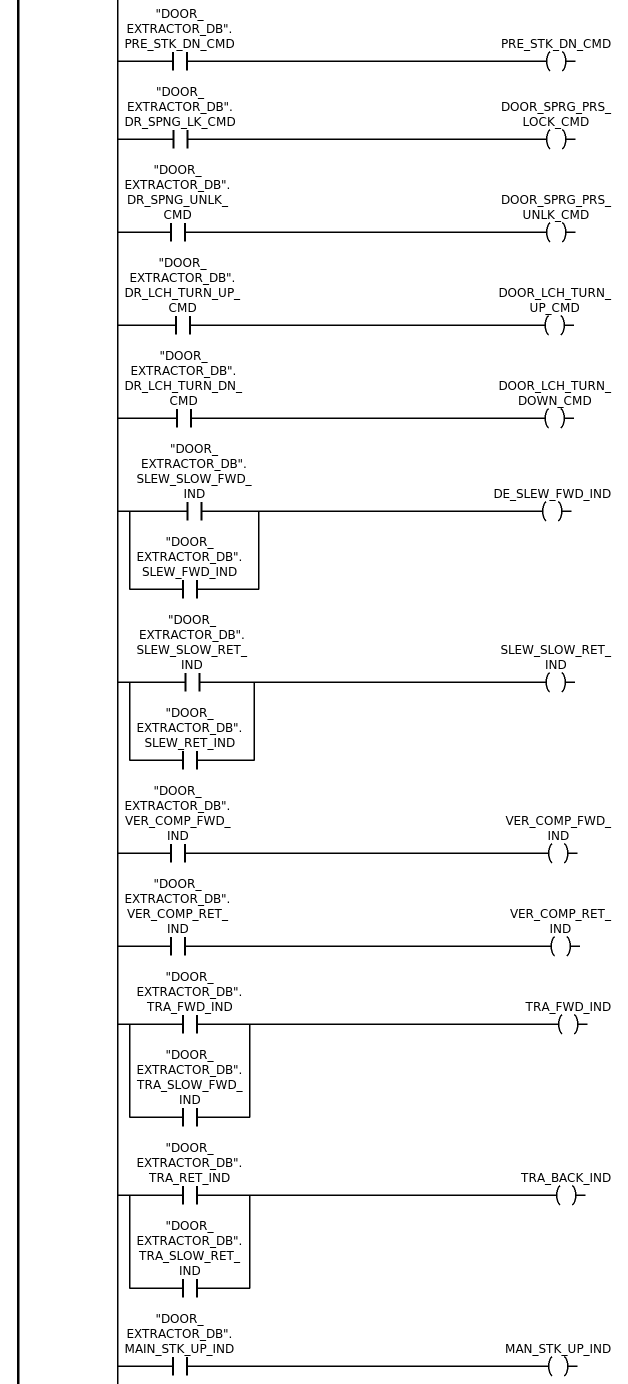
[picture p48: OUTPUT_MAPPING networks 12-12]
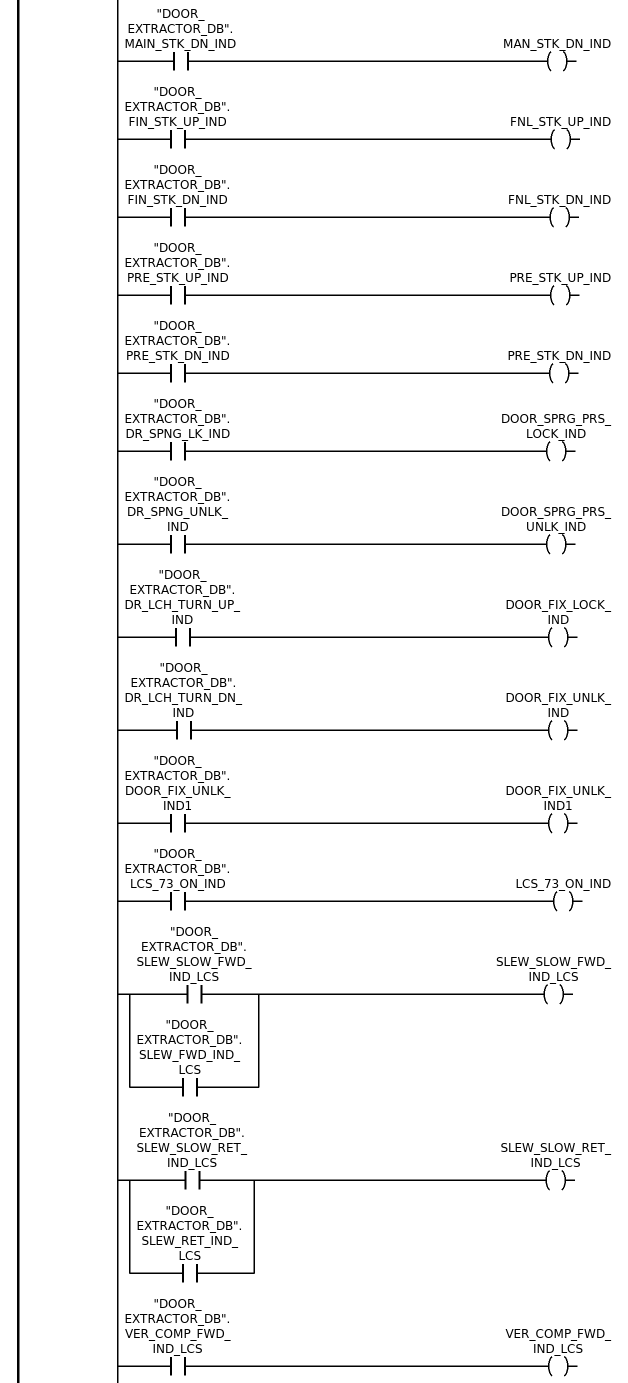
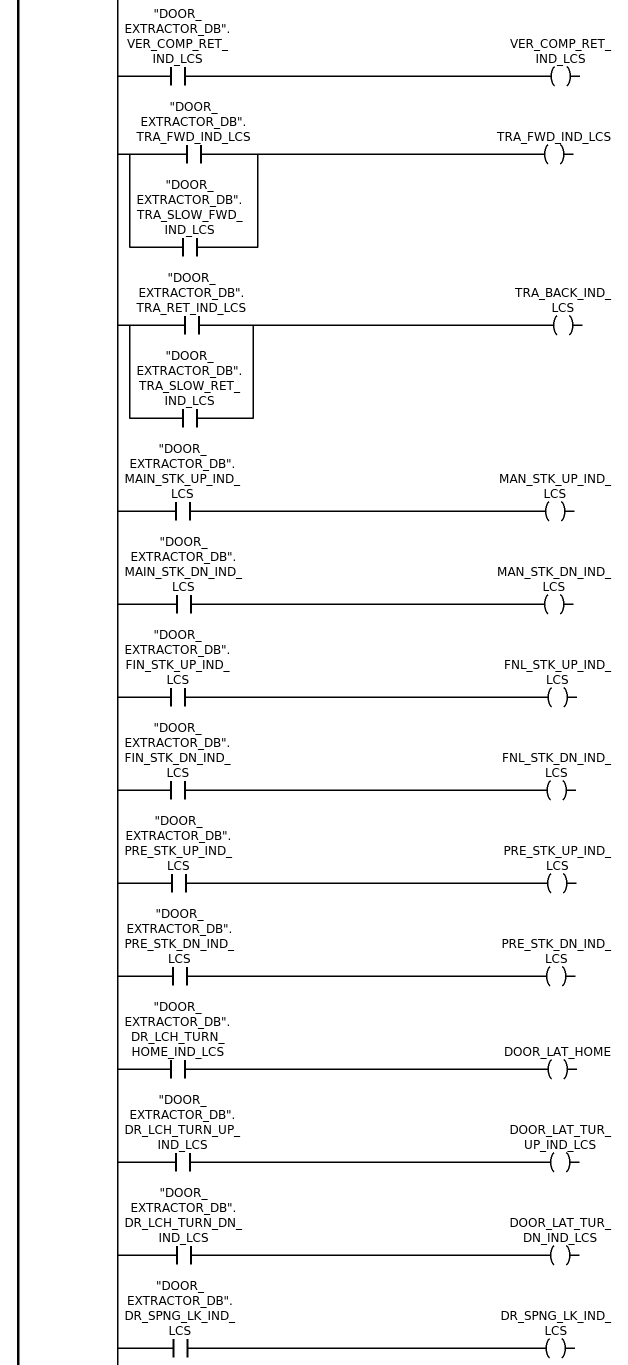
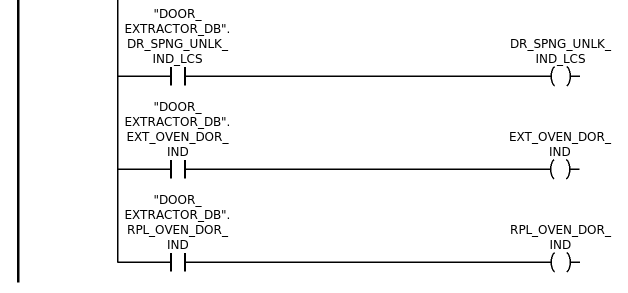
NETWORK
TITLE =
      A     "ALWAYS_ON";
      =     L 0.0;
      A     L 0.0;
      A     "DOOR_EXTRACTOR_DB".SLEW_NOR_FWD_COMMAND;
      =     "SLEW_NOR_FWD_COMMAND";
      A     L 0.0;
      A     "DOOR_EXTRACTOR_DB".SLEW_NOR_RET_COMMAND;
      =     "SLEW_NOR_RET_COMMAND";
      A     L 0.0;
      A     "DOOR_EXTRACTOR_DB".VER_COMP_FWD_CMD;
      =     "VER_COMP_FWD_CMD";
      A     L 0.0;
      A     "DOOR_EXTRACTOR_DB".VER_COMP_RET_CMD;
      =     "VER_COMP_RET_CMD";
      A     L 0.0;
      A     "DOOR_EXTRACTOR_DB".VER_COMP_RELIVE_CMD;
      =     "VER_COMP_RELIVE_CMD";
      A     L 0.0;
      A     "DOOR_EXTRACTOR_DB".TRA_SLOW_FWD_CMD;
      =     "TRA_SLOW_FWD_CMD";
      A     L 0.0;
      A     "DOOR_EXTRACTOR_DB".TRA_SLOW_RET_CMD;
      =     "TRA_SLOW_RET_CMD";
      A     L 0.0;
      A     "DOOR_EXTRACTOR_DB".TRA_NOR_FWD_CMD;
      =     "TRA_NORM_FWD_CMD";
      A     L 0.0;
      A     "DOOR_EXTRACTOR_DB".TRA_NOR_RET_CMD;
      =     "TRA_NORM_RET_CMD";
      A     L 0.0;
      A     "DOOR_EXTRACTOR_DB".TRA_RELIVE_CMD;
      =     "DE_TRA_RELIVE_CMD";
      A     L 0.0;
      A(;
      O     "DOOR_EXTRACTOR_DB".MAIN_STK_UP_CMD;
      O     "DOOR_EXTRACTOR_DB".FIN_STK_UP_CMD;
      );
      =     "MAN_FNL_STK_UP_CMD";
      A     L 0.0;
      A(;
      O     "DOOR_EXTRACTOR_DB".MAIN_STK_DN_CMD;
      O     "DOOR_EXTRACTOR_DB".FIN_STK_DN_CMD;
      );
      =     "MAN_FNL_STK_DN_CMD";
      A     L 0.0;
      A     "DOOR_EXTRACTOR_DB".PRE_STK_UP_CMD;
      =     "PRE_STK_UP_CMD";
      A     L 0.0;
      A     "DOOR_EXTRACTOR_DB".PRE_STK_DN_CMD;
      =     "PRE_STK_DN_CMD";
      A     L 0.0;
      A     "DOOR_EXTRACTOR_DB".DR_SPNG_LK_CMD;
      =     "DOOR_SPRG_PRS_LOCK_CMD";
      A     L 0.0;
      A     "DOOR_EXTRACTOR_DB".DR_SPNG_UNLK_CMD;
      =     "DOOR_SPRG_PRS_UNLK_CMD";
      A     L 0.0;
      A     "DOOR_EXTRACTOR_DB".DR_LCH_TURN_UP_CMD;
      =     "DOOR_LCH_TURN_UP_CMD";
      A     L 0.0;
      A     "DOOR_EXTRACTOR_DB".DR_LCH_TURN_DN_CMD;
      =     "DOOR_LCH_TURN_DOWN_CMD";
      A     L 0.0;
      A(;
      O     "DOOR_EXTRACTOR_DB".SLEW_SLOW_FWD_IND;
      O     "DOOR_EXTRACTOR_DB".SLEW_FWD_IND;
      );
      =     "DE_SLEW_FWD_IND";
      A     L 0.0;
      A(;
      O     "DOOR_EXTRACTOR_DB".SLEW_SLOW_RET_IND;
      O     "DOOR_EXTRACTOR_DB".SLEW_RET_IND;
      );
      =     "SLEW_SLOW_RET_IND";
      A     L 0.0;
      A     "DOOR_EXTRACTOR_DB".VER_COMP_FWD_IND;
      =     "VER_COMP_FWD_IND";
      A     L 0.0;
      A     "DOOR_EXTRACTOR_DB".VER_COMP_RET_IND;
      =     "VER_COMP_RET_IND";
      A     L 0.0;
      A(;
      O     "DOOR_EXTRACTOR_DB".TRA_FWD_IND;
      O     "DOOR_EXTRACTOR_DB".TRA_SLOW_FWD_IND;
      );
      =     "TRA_FWD_IND";
      A     L 0.0;
      A(;
      O     "DOOR_EXTRACTOR_DB".TRA_RET_IND;
      O     "DOOR_EXTRACTOR_DB".TRA_SLOW_RET_IND;
      );
      =     "TRA_BACK_IND";
      A     L 0.0;
      A     "DOOR_EXTRACTOR_DB".MAIN_STK_UP_IND;
      =     "MAN_STK_UP_IND";
      A     L 0.0;
      A     "DOOR_EXTRACTOR_DB".MAIN_STK_DN_IND;
      =     "MAN_STK_DN_IND";
      A     L 0.0;
      A     "DOOR_EXTRACTOR_DB".FIN_STK_UP_IND;
      =     "FNL_STK_UP_IND";
      A     L 0.0;
      A     "DOOR_EXTRACTOR_DB".FIN_STK_DN_IND;
      =     "FNL_STK_DN_IND";
      A     L 0.0;
      A     "DOOR_EXTRACTOR_DB".PRE_STK_UP_IND;
      =     "PRE_STK_UP_IND";
      A     L 0.0;
      A     "DOOR_EXTRACTOR_DB".PRE_STK_DN_IND;
      =     "PRE_STK_DN_IND";
      A     L 0.0;
      A     "DOOR_EXTRACTOR_DB".DR_SPNG_LK_IND;
      =     "DOOR_SPRG_PRS_LOCK_IND";
      A     L 0.0;
      A     "DOOR_EXTRACTOR_DB".DR_SPNG_UNLK_IND;
      =     "DOOR_SPRG_PRS_UNLK_IND";
      A     L 0.0;
      A     "DOOR_EXTRACTOR_DB".DR_LCH_TURN_UP_IND;
      =     "DOOR_FIX_LOCK_IND";
      A     L 0.0;
      A     "DOOR_EXTRACTOR_DB".DR_LCH_TURN_DN_IND;
      =     "DOOR_FIX_UNLK_IND";
      A     L 0.0;
      A     "DOOR_EXTRACTOR_DB".DOOR_FIX_UNLK_IND1;
      =     "DOOR_FIX_UNLK_IND1";
      A     L 0.0;
      A     "DOOR_EXTRACTOR_DB".LCS_73_ON_IND;
      =     "LCS_73_ON_IND";
      A     L 0.0;
      A(;
      O     "DOOR_EXTRACTOR_DB".SLEW_SLOW_FWD_IND_LCS;
      O     "DOOR_EXTRACTOR_DB".SLEW_FWD_IND_LCS;
      );
      =     "SLEW_SLOW_FWD_IND_LCS";
      A     L 0.0;
      A(;
      O     "DOOR_EXTRACTOR_DB".SLEW_SLOW_RET_IND_LCS;
      O     "DOOR_EXTRACTOR_DB".SLEW_RET_IND_LCS;
      );
      =     "SLEW_SLOW_RET_IND_LCS";
      A     L 0.0;
      A     "DOOR_EXTRACTOR_DB".VER_COMP_FWD_IND_LCS;
      =     "VER_COMP_FWD_IND_LCS";
      A     L 0.0;
      A     "DOOR_EXTRACTOR_DB".VER_COMP_RET_IND_LCS;
      =     "VER_COMP_RET_IND_LCS";
      A     L 0.0;
      A(;
      O     "DOOR_EXTRACTOR_DB".TRA_FWD_IND_LCS;
      O     "DOOR_EXTRACTOR_DB".TRA_SLOW_FWD_IND_LCS;
      );
      =     "TRA_FWD_IND_LCS";
      A     L 0.0;
      A(;
      O     "DOOR_EXTRACTOR_DB".TRA_RET_IND_LCS;
      O     "DOOR_EXTRACTOR_DB".TRA_SLOW_RET_IND_LCS;
      );
      =     "TRA_BACK_IND_LCS";
      A     L 0.0;
      A     "DOOR_EXTRACTOR_DB".MAIN_STK_UP_IND_LCS;
      =     "MAN_STK_UP_IND_LCS";
      A     L 0.0;
      A     "DOOR_EXTRACTOR_DB".MAIN_STK_DN_IND_LCS;
      =     "MAN_STK_DN_IND_LCS";
      A     L 0.0;
      A     "DOOR_EXTRACTOR_DB".FIN_STK_UP_IND_LCS;
      =     "FNL_STK_UP_IND_LCS";
      A     L 0.0;
      A     "DOOR_EXTRACTOR_DB".FIN_STK_DN_IND_LCS;
      =     "FNL_STK_DN_IND_LCS";
      A     L 0.0;
      A     "DOOR_EXTRACTOR_DB".PRE_STK_UP_IND_LCS;
      =     "PRE_STK_UP_IND_LCS";
      A     L 0.0;
      A     "DOOR_EXTRACTOR_DB".PRE_STK_DN_IND_LCS;
      =     "PRE_STK_DN_IND_LCS";
      A     L 0.0;
      A     "DOOR_EXTRACTOR_DB".DR_LCH_TURN_HOME_IND_LCS;
      =     "DOOR_LAT_HOME";
      A     L 0.0;
      A     "DOOR_EXTRACTOR_DB".DR_LCH_TURN_UP_IND_LCS;
      =     "DOOR_LAT_TUR_UP_IND_LCS";
      A     L 0.0;
      A     "DOOR_EXTRACTOR_DB".DR_LCH_TURN_DN_IND_LCS;
      =     "DOOR_LAT_TUR_DN_IND_LCS";
      A     L 0.0;
      A     "DOOR_EXTRACTOR_DB".DR_SPNG_LK_IND_LCS;
      =     "DR_SPNG_LK_IND_LCS";
      A     L 0.0;
      A     "DOOR_EXTRACTOR_DB".DR_SPNG_UNLK_IND_LCS;
      =     "DR_SPNG_UNLK_IND_LCS";
      A     L 0.0;
      A     "DOOR_EXTRACTOR_DB".EXT_OVEN_DOR_IND;
      =     "EXT_OVEN_DOR_IND";
      A     L 0.0;
      A     "DOOR_EXTRACTOR_DB".RPL_OVEN_DOR_IND;
      =     "RPL_OVEN_DOR_IND";
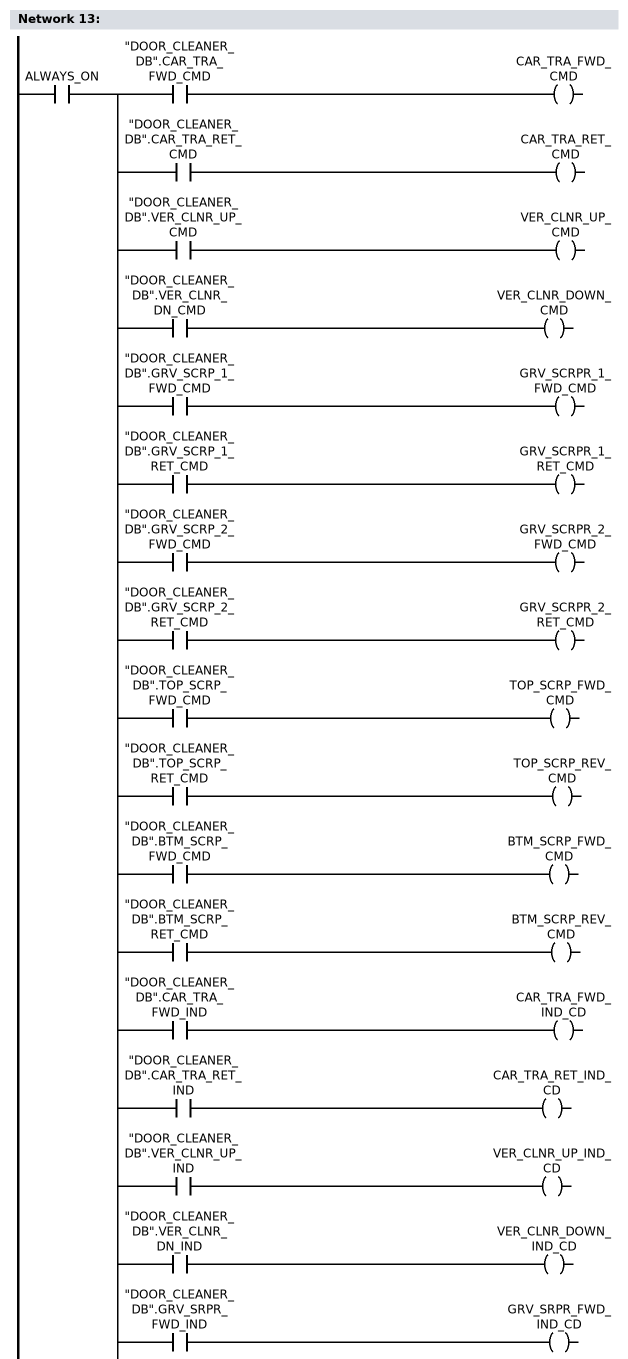
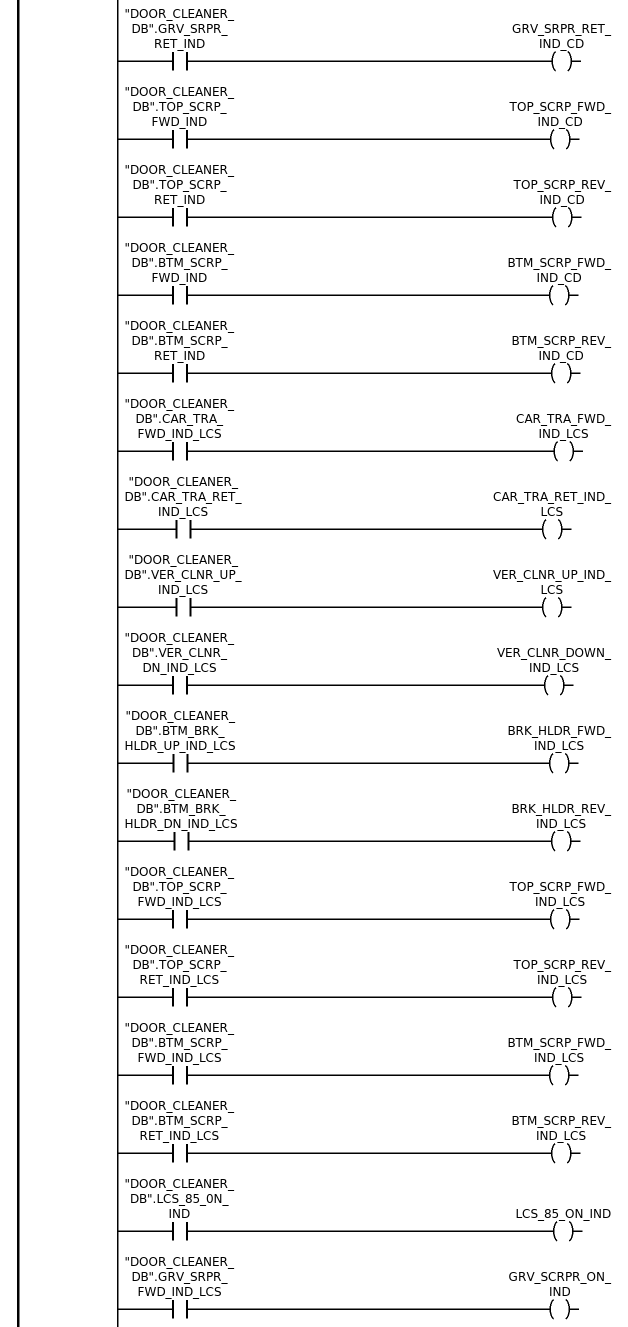
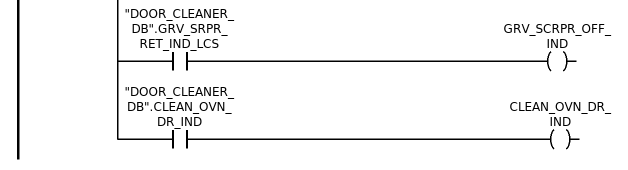
NETWORK
TITLE =
      A     "ALWAYS_ON";
      =     L 0.0;
      A     L 0.0;
      A     "DOOR_CLEANER_DB".CAR_TRA_FWD_CMD;
      =     "CAR_TRA_FWD_CMD";
      A     L 0.0;
      A     "DOOR_CLEANER_DB".CAR_TRA_RET_CMD;
      =     "CAR_TRA_RET_CMD";
      A     L 0.0;
      A     "DOOR_CLEANER_DB".VER_CLNR_UP_CMD;
      =     "VER_CLNR_UP_CMD";
      A     L 0.0;
      A     "DOOR_CLEANER_DB".VER_CLNR_DN_CMD;
      =     "VER_CLNR_DOWN_CMD";
      A     L 0.0;
      A     "DOOR_CLEANER_DB".GRV_SCRP_1_FWD_CMD;
      =     "GRV_SCRPR_1_FWD_CMD";
      A     L 0.0;
      A     "DOOR_CLEANER_DB".GRV_SCRP_1_RET_CMD;
      =     "GRV_SCRPR_1_RET_CMD";
      A     L 0.0;
      A     "DOOR_CLEANER_DB".GRV_SCRP_2_FWD_CMD;
      =     "GRV_SCRPR_2_FWD_CMD";
      A     L 0.0;
      A     "DOOR_CLEANER_DB".GRV_SCRP_2_RET_CMD;
      =     "GRV_SCRPR_2_RET_CMD";
      A     L 0.0;
      A     "DOOR_CLEANER_DB".TOP_SCRP_FWD_CMD;
      =     "TOP_SCRP_FWD_CMD";
      A     L 0.0;
      A     "DOOR_CLEANER_DB".TOP_SCRP_RET_CMD;
      =     "TOP_SCRP_REV_CMD";
      A     L 0.0;
      A     "DOOR_CLEANER_DB".BTM_SCRP_FWD_CMD;
      =     "BTM_SCRP_FWD_CMD";
      A     L 0.0;
      A     "DOOR_CLEANER_DB".BTM_SCRP_RET_CMD;
      =     "BTM_SCRP_REV_CMD";
      A     L 0.0;
      A     "DOOR_CLEANER_DB".CAR_TRA_FWD_IND;
      =     "CAR_TRA_FWD_IND_CD";
      A     L 0.0;
      A     "DOOR_CLEANER_DB".CAR_TRA_RET_IND;
      =     "CAR_TRA_RET_IND_CD";
      A     L 0.0;
      A     "DOOR_CLEANER_DB".VER_CLNR_UP_IND;
      =     "VER_CLNR_UP_IND_CD";
      A     L 0.0;
      A     "DOOR_CLEANER_DB".VER_CLNR_DN_IND;
      =     "VER_CLNR_DOWN_IND_CD";
      A     L 0.0;
      A     "DOOR_CLEANER_DB".GRV_SRPR_FWD_IND;
      =     "GRV_SRPR_FWD_IND_CD";
      A     L 0.0;
      A     "DOOR_CLEANER_DB".GRV_SRPR_RET_IND;
      =     "GRV_SRPR_RET_IND_CD";
      A     L 0.0;
      A     "DOOR_CLEANER_DB".TOP_SCRP_FWD_IND;
      =     "TOP_SCRP_FWD_IND_CD";
      A     L 0.0;
      A     "DOOR_CLEANER_DB".TOP_SCRP_RET_IND;
      =     "TOP_SCRP_REV_IND_CD";
      A     L 0.0;
      A     "DOOR_CLEANER_DB".BTM_SCRP_FWD_IND;
      =     "BTM_SCRP_FWD_IND_CD";
      A     L 0.0;
      A     "DOOR_CLEANER_DB".BTM_SCRP_RET_IND;
      =     "BTM_SCRP_REV_IND_CD";
      A     L 0.0;
      A     "DOOR_CLEANER_DB".CAR_TRA_FWD_IND_LCS;
      =     "CAR_TRA_FWD_IND_LCS";
      A     L 0.0;
      A     "DOOR_CLEANER_DB".CAR_TRA_RET_IND_LCS;
      =     "CAR_TRA_RET_IND_LCS";
      A     L 0.0;
      A     "DOOR_CLEANER_DB".VER_CLNR_UP_IND_LCS;
      =     "VER_CLNR_UP_IND_LCS";
      A     L 0.0;
      A     "DOOR_CLEANER_DB".VER_CLNR_DN_IND_LCS;
      =     "VER_CLNR_DOWN_IND_LCS";
      A     L 0.0;
      A     "DOOR_CLEANER_DB".BTM_BRK_HLDR_UP_IND_LCS;
      =     "BRK_HLDR_FWD_IND_LCS";
      A     L 0.0;
      A     "DOOR_CLEANER_DB".BTM_BRK_HLDR_DN_IND_LCS;
      =     "BRK_HLDR_REV_IND_LCS";
      A     L 0.0;
      A     "DOOR_CLEANER_DB".TOP_SCRP_FWD_IND_LCS;
      =     "TOP_SCRP_FWD_IND_LCS";
      A     L 0.0;
      A     "DOOR_CLEANER_DB".TOP_SCRP_RET_IND_LCS;
      =     "TOP_SCRP_REV_IND_LCS";
      A     L 0.0;
      A     "DOOR_CLEANER_DB".BTM_SCRP_FWD_IND_LCS;
      =     "BTM_SCRP_FWD_IND_LCS";
      A     L 0.0;
      A     "DOOR_CLEANER_DB".BTM_SCRP_RET_IND_LCS;
      =     "BTM_SCRP_REV_IND_LCS";
      A     L 0.0;
      A     "DOOR_CLEANER_DB".LCS_85_0N_IND;
      =     "LCS_85_ON_IND";
      A     L 0.0;
      A     "DOOR_CLEANER_DB".GRV_SRPR_FWD_IND_LCS;
      =     "GRV_SCRPR_ON_IND";
      A     L 0.0;
      A     "DOOR_CLEANER_DB".GRV_SRPR_RET_IND_LCS;
      =     "GRV_SCRPR_OFF_IND";
      A     L 0.0;
      A     "DOOR_CLEANER_DB".CLEAN_OVN_DR_IND;
      =     "CLEAN_OVN_DR_IND";
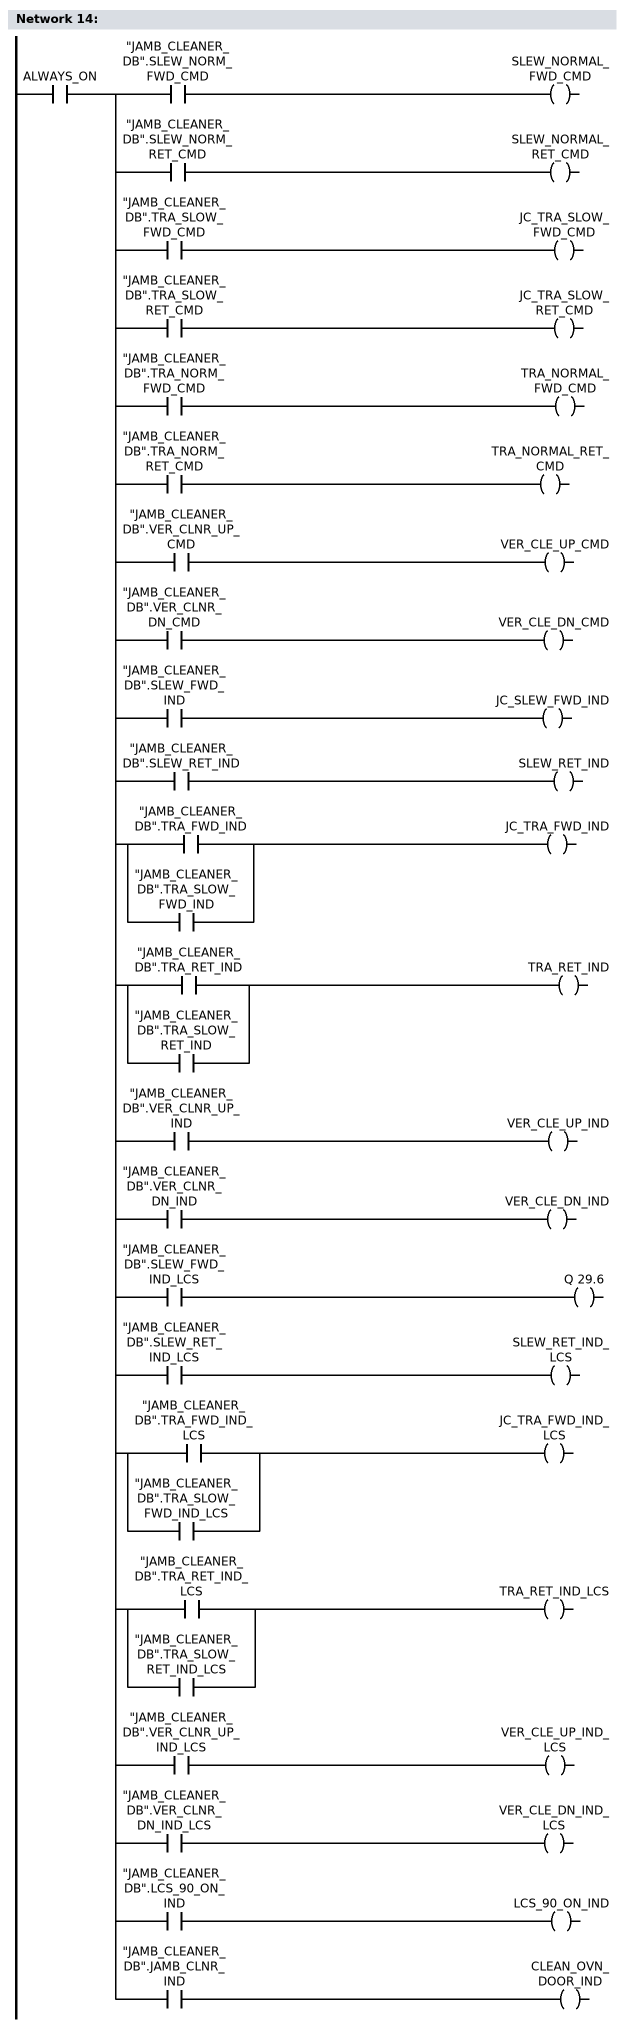
NETWORK
TITLE =
      A     "ALWAYS_ON";
      =     L 0.0;
      A     L 0.0;
      A     "JAMB_CLEANER_DB".SLEW_NORM_FWD_CMD;
      =     "SLEW_NORMAL_FWD_CMD";
      A     L 0.0;
      A     "JAMB_CLEANER_DB".SLEW_NORM_RET_CMD;
      =     "SLEW_NORMAL_RET_CMD";
      A     L 0.0;
      A     "JAMB_CLEANER_DB".TRA_SLOW_FWD_CMD;
      =     "JC_TRA_SLOW_FWD_CMD";
      A     L 0.0;
      A     "JAMB_CLEANER_DB".TRA_SLOW_RET_CMD;
      =     "JC_TRA_SLOW_RET_CMD";
      A     L 0.0;
      A     "JAMB_CLEANER_DB".TRA_NORM_FWD_CMD;
      =     "TRA_NORMAL_FWD_CMD";
      A     L 0.0;
      A     "JAMB_CLEANER_DB".TRA_NORM_RET_CMD;
      =     "TRA_NORMAL_RET_CMD";
      A     L 0.0;
      A     "JAMB_CLEANER_DB".VER_CLNR_UP_CMD;
      =     "VER_CLE_UP_CMD";
      A     L 0.0;
      A     "JAMB_CLEANER_DB".VER_CLNR_DN_CMD;
      =     "VER_CLE_DN_CMD";
      A     L 0.0;
      A     "JAMB_CLEANER_DB".SLEW_FWD_IND;
      =     "JC_SLEW_FWD_IND";
      A     L 0.0;
      A     "JAMB_CLEANER_DB".SLEW_RET_IND;
      =     "SLEW_RET_IND";
      A     L 0.0;
      A(;
      O     "JAMB_CLEANER_DB".TRA_FWD_IND;
      O     "JAMB_CLEANER_DB".TRA_SLOW_FWD_IND;
      );
      =     "JC_TRA_FWD_IND";
      A     L 0.0;
      A(;
      O     "JAMB_CLEANER_DB".TRA_RET_IND;
      O     "JAMB_CLEANER_DB".TRA_SLOW_RET_IND;
      );
      =     "TRA_RET_IND";
      A     L 0.0;
      A     "JAMB_CLEANER_DB".VER_CLNR_UP_IND;
      =     "VER_CLE_UP_IND";
      A     L 0.0;
      A     "JAMB_CLEANER_DB".VER_CLNR_DN_IND;
      =     "VER_CLE_DN_IND";
      A     L 0.0;
      A     "JAMB_CLEANER_DB".SLEW_FWD_IND_LCS;
      =     Q 29.6;
      A     L 0.0;
      A     "JAMB_CLEANER_DB".SLEW_RET_IND_LCS;
      =     "SLEW_RET_IND_LCS";
      A     L 0.0;
      A(;
      O     "JAMB_CLEANER_DB".TRA_FWD_IND_LCS;
      O     "JAMB_CLEANER_DB".TRA_SLOW_FWD_IND_LCS;
      );
      =     "JC_TRA_FWD_IND_LCS";
      A     L 0.0;
      A(;
      O     "JAMB_CLEANER_DB".TRA_RET_IND_LCS;
      O     "JAMB_CLEANER_DB".TRA_SLOW_RET_IND_LCS;
      );
      =     "TRA_RET_IND_LCS";
      A     L 0.0;
      A     "JAMB_CLEANER_DB".VER_CLNR_UP_IND_LCS;
      =     "VER_CLE_UP_IND_LCS";
      A     L 0.0;
      A     "JAMB_CLEANER_DB".VER_CLNR_DN_IND_LCS;
      =     "VER_CLE_DN_IND_LCS";
      A     L 0.0;
      A     "JAMB_CLEANER_DB".LCS_90_ON_IND;
      =     "LCS_90_ON_IND";
      A     L 0.0;
      A     "JAMB_CLEANER_DB".JAMB_CLNR_IND;
      =     "CLEAN_OVN_DOOR_IND";
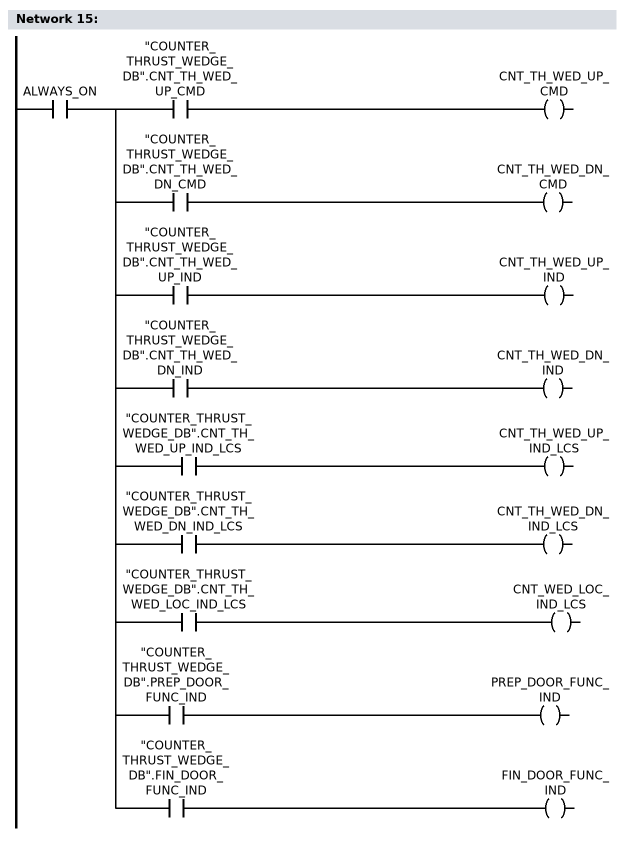
NETWORK
TITLE =
      A     "ALWAYS_ON";
      =     L 0.0;
      A     L 0.0;
      A     "COUNTER_THRUST_WEDGE_DB".CNT_TH_WED_UP_CMD;
      =     "CNT_TH_WED_UP_CMD";
      A     L 0.0;
      A     "COUNTER_THRUST_WEDGE_DB".CNT_TH_WED_DN_CMD;
      =     "CNT_TH_WED_DN_CMD";
      A     L 0.0;
      A     "COUNTER_THRUST_WEDGE_DB".CNT_TH_WED_UP_IND;
      =     "CNT_TH_WED_UP_IND";
      A     L 0.0;
      A     "COUNTER_THRUST_WEDGE_DB".CNT_TH_WED_DN_IND;
      =     "CNT_TH_WED_DN_IND";
      A     L 0.0;
      A     "COUNTER_THRUST_WEDGE_DB".CNT_TH_WED_UP_IND_LCS;
      =     "CNT_TH_WED_UP_IND_LCS";
      A     L 0.0;
      A     "COUNTER_THRUST_WEDGE_DB".CNT_TH_WED_DN_IND_LCS;
      =     "CNT_TH_WED_DN_IND_LCS";
      A     L 0.0;
      A     "COUNTER_THRUST_WEDGE_DB".CNT_TH_WED_LOC_IND_LCS;
      =     "CNT_WED_LOC_IND_LCS";
      A     L 0.0;
      A     "COUNTER_THRUST_WEDGE_DB".PREP_DOOR_FUNC_IND;
      =     "PREP_DOOR_FUNC_IND";
      A     L 0.0;
      A     "COUNTER_THRUST_WEDGE_DB".FIN_DOOR_FUNC_IND;
      =     "FIN_DOOR_FUNC_IND";
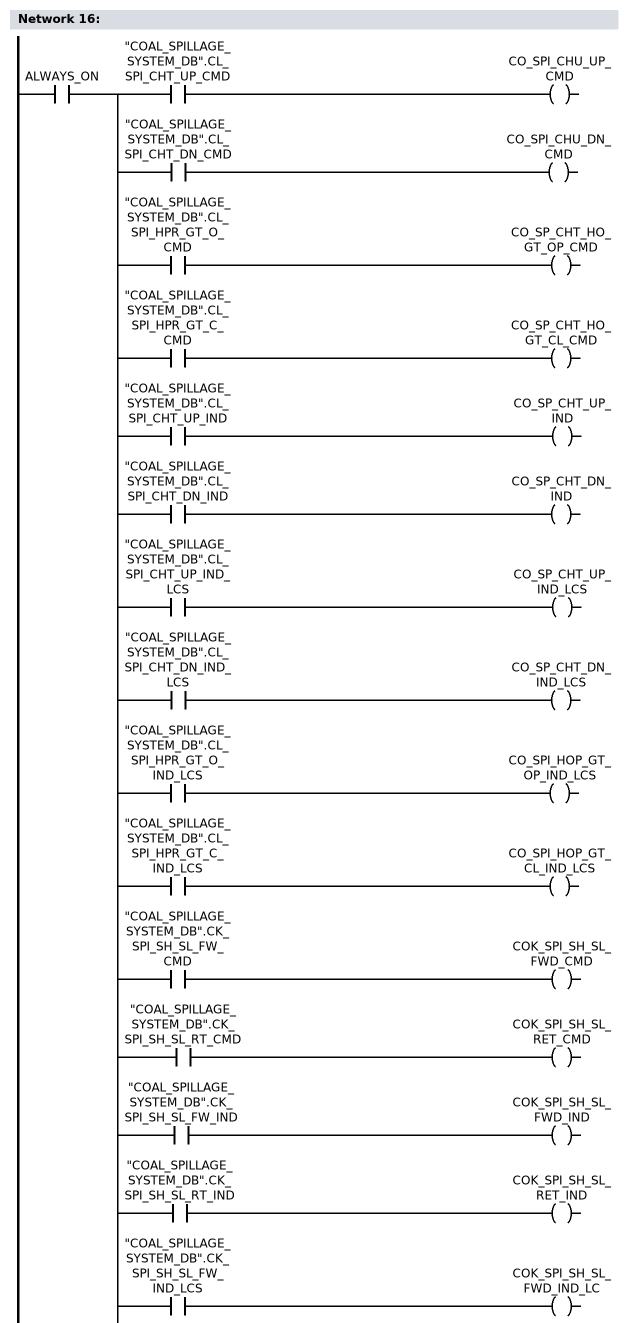
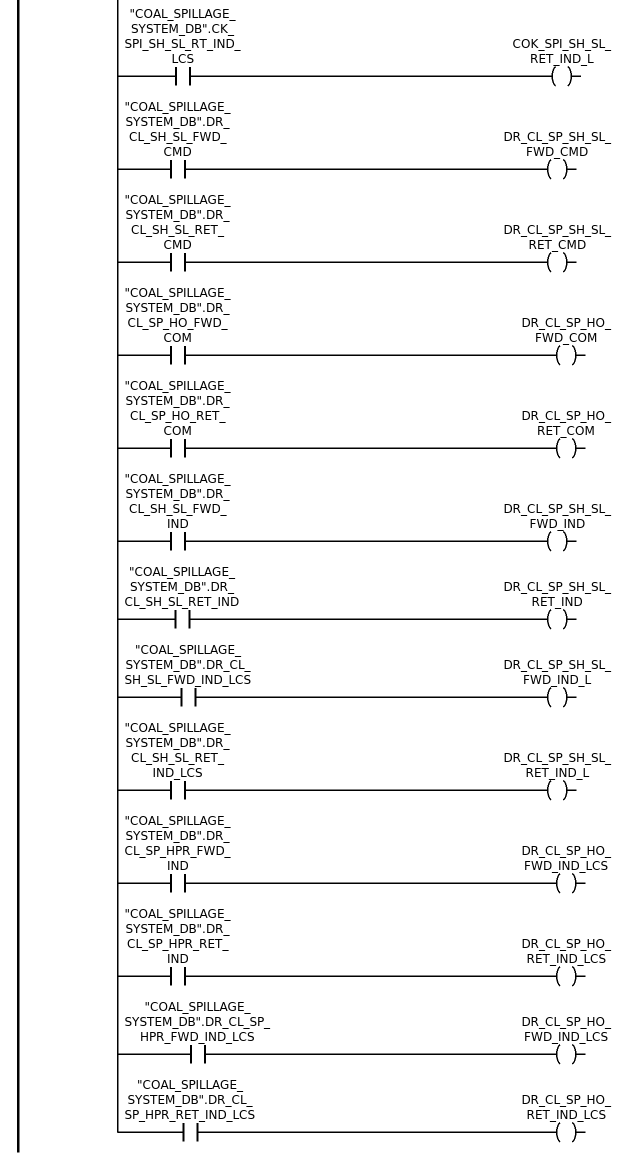
NETWORK
TITLE =
      A     "ALWAYS_ON";
      =     L 0.0;
      A     L 0.0;
      A     "COAL_SPILLAGE_SYSTEM_DB".CL_SPI_CHT_UP_CMD;
      =     "CO_SPI_CHU_UP_CMD";
      A     L 0.0;
      A     "COAL_SPILLAGE_SYSTEM_DB".CL_SPI_CHT_DN_CMD;
      =     "CO_SPI_CHU_DN_CMD";
      A     L 0.0;
      A     "COAL_SPILLAGE_SYSTEM_DB".CL_SPI_HPR_GT_O_CMD;
      =     "CO_SP_CHT_HO_GT_OP_CMD";
      A     L 0.0;
      A     "COAL_SPILLAGE_SYSTEM_DB".CL_SPI_HPR_GT_C_CMD;
      =     "CO_SP_CHT_HO_GT_CL_CMD";
      A     L 0.0;
      A     "COAL_SPILLAGE_SYSTEM_DB".CL_SPI_CHT_UP_IND;
      =     "CO_SP_CHT_UP_IND";
      A     L 0.0;
      A     "COAL_SPILLAGE_SYSTEM_DB".CL_SPI_CHT_DN_IND;
      =     "CO_SP_CHT_DN_IND";
      A     L 0.0;
      A     "COAL_SPILLAGE_SYSTEM_DB".CL_SPI_CHT_UP_IND_LCS;
      =     "CO_SP_CHT_UP_IND_LCS";
      A     L 0.0;
      A     "COAL_SPILLAGE_SYSTEM_DB".CL_SPI_CHT_DN_IND_LCS;
      =     "CO_SP_CHT_DN_IND_LCS";
      A     L 0.0;
      A     "COAL_SPILLAGE_SYSTEM_DB".CL_SPI_HPR_GT_O_IND_LCS;
      =     "CO_SPI_HOP_GT_OP_IND_LCS";
      A     L 0.0;
      A     "COAL_SPILLAGE_SYSTEM_DB".CL_SPI_HPR_GT_C_IND_LCS;
      =     "CO_SPI_HOP_GT_CL_IND_LCS";
      A     L 0.0;
      A     "COAL_SPILLAGE_SYSTEM_DB".CK_SPI_SH_SL_FW_CMD;
      =     "COK_SPI_SH_SL_FWD_CMD";
      A     L 0.0;
      A     "COAL_SPILLAGE_SYSTEM_DB".CK_SPI_SH_SL_RT_CMD;
      =     "COK_SPI_SH_SL_RET_CMD";
      A     L 0.0;
      A     "COAL_SPILLAGE_SYSTEM_DB".CK_SPI_SH_SL_FW_IND;
      =     "COK_SPI_SH_SL_FWD_IND";
      A     L 0.0;
      A     "COAL_SPILLAGE_SYSTEM_DB".CK_SPI_SH_SL_RT_IND;
      =     "COK_SPI_SH_SL_RET_IND";
      A     L 0.0;
      A     "COAL_SPILLAGE_SYSTEM_DB".CK_SPI_SH_SL_FW_IND_LCS;
      =     "COK_SPI_SH_SL_FWD_IND_LC";
      A     L 0.0;
      A     "COAL_SPILLAGE_SYSTEM_DB".CK_SPI_SH_SL_RT_IND_LCS;
      =     "COK_SPI_SH_SL_RET_IND_L";
      A     L 0.0;
      A     "COAL_SPILLAGE_SYSTEM_DB".DR_CL_SH_SL_FWD_CMD;
      =     "DR_CL_SP_SH_SL_FWD_CMD";
      A     L 0.0;
      A     "COAL_SPILLAGE_SYSTEM_DB".DR_CL_SH_SL_RET_CMD;
      =     "DR_CL_SP_SH_SL_RET_CMD";
      A     L 0.0;
      A     "COAL_SPILLAGE_SYSTEM_DB".DR_CL_SP_HO_FWD_COM;
      =     "DR_CL_SP_HO_FWD_COM";
      A     L 0.0;
      A     "COAL_SPILLAGE_SYSTEM_DB".DR_CL_SP_HO_RET_COM;
      =     "DR_CL_SP_HO_RET_COM";
      A     L 0.0;
      A     "COAL_SPILLAGE_SYSTEM_DB".DR_CL_SH_SL_FWD_IND;
      =     "DR_CL_SP_SH_SL_FWD_IND";
      A     L 0.0;
      A     "COAL_SPILLAGE_SYSTEM_DB".DR_CL_SH_SL_RET_IND;
      =     "DR_CL_SP_SH_SL_RET_IND";
      A     L 0.0;
      A     "COAL_SPILLAGE_SYSTEM_DB".DR_CL_SH_SL_FWD_IND_LCS;
      =     "DR_CL_SP_SH_SL_FWD_IND_L";
      A     L 0.0;
      A     "COAL_SPILLAGE_SYSTEM_DB".DR_CL_SH_SL_RET_IND_LCS;
      =     "DR_CL_SP_SH_SL_RET_IND_L";
      A     L 0.0;
      A     "COAL_SPILLAGE_SYSTEM_DB".DR_CL_SP_HPR_FWD_IND;
      =     "DR_CL_SP_HO_FWD_IND_LCS";
      A     L 0.0;
      A     "COAL_SPILLAGE_SYSTEM_DB".DR_CL_SP_HPR_RET_IND;
      =     "DR_CL_SP_HO_RET_IND_LCS";
      A     L 0.0;
      A     "COAL_SPILLAGE_SYSTEM_DB".DR_CL_SP_HPR_FWD_IND_LCS;
      =     "DR_CL_SP_HO_FWD_IND_LCS";
      A     L 0.0;
      A     "COAL_SPILLAGE_SYSTEM_DB".DR_CL_SP_HPR_RET_IND_LCS;
      =     "DR_CL_SP_HO_RET_IND_LCS";
END_FUNCTION

FUNCTION "MAIN_POWER" : VOID	// FC 3
AUTHOR : Kamillas
VERSION : 0.1
BEGIN
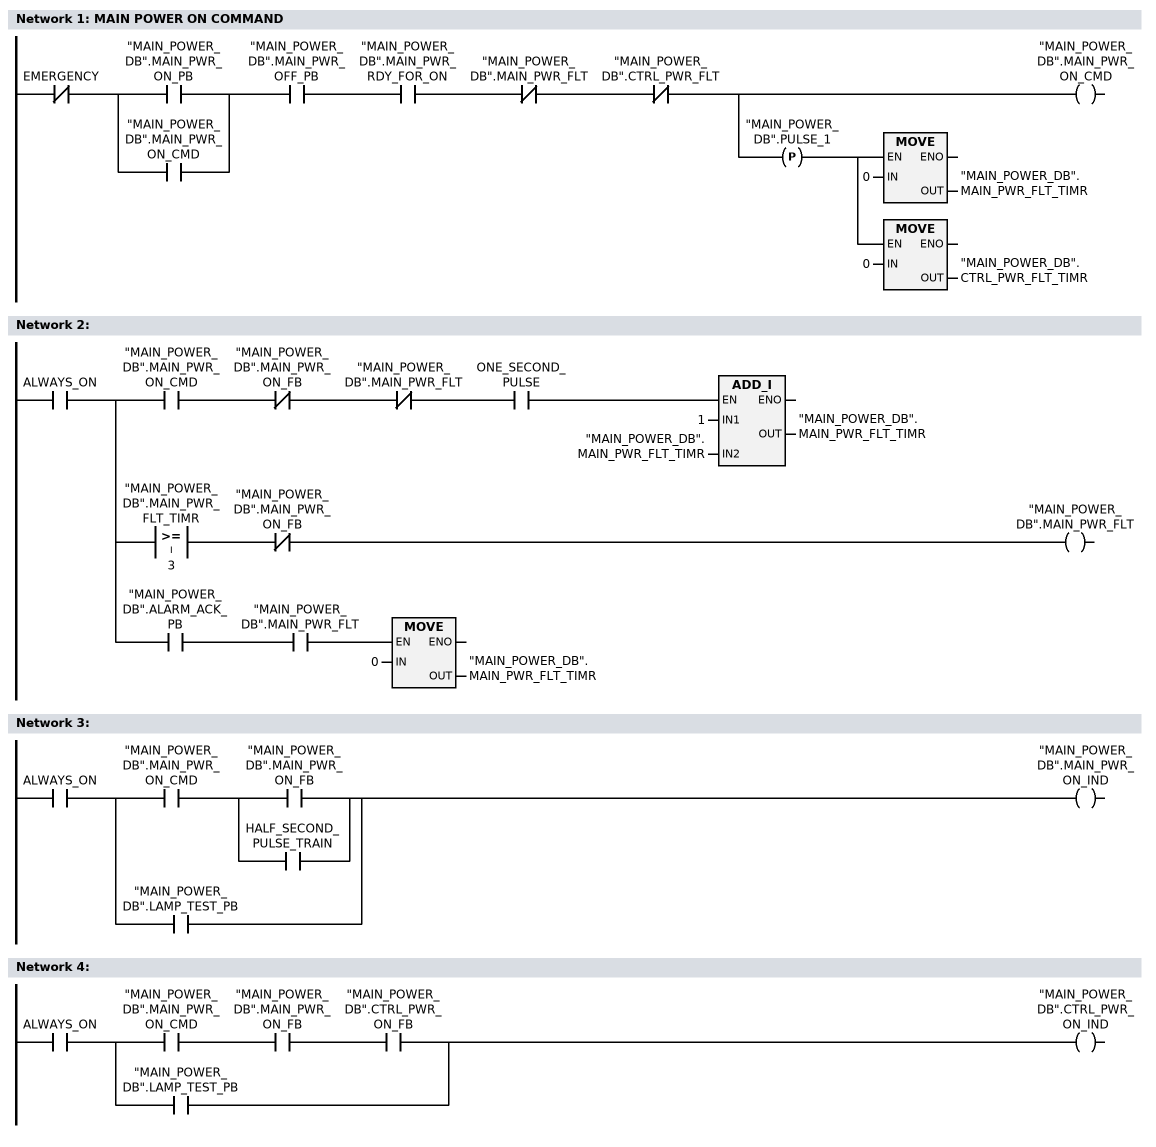
NETWORK
TITLE = MAIN POWER ON COMMAND
      AN    "EMERGENCY";
      A(;
      O     "MAIN_POWER_DB".MAIN_PWR_ON_PB;
      O     "MAIN_POWER_DB".MAIN_PWR_ON_CMD;
      );
      A     "MAIN_POWER_DB".MAIN_PWR_OFF_PB;
      A     "MAIN_POWER_DB".MAIN_PWR_RDY_FOR_ON;
      AN    "MAIN_POWER_DB".MAIN_PWR_FLT;
      AN    "MAIN_POWER_DB".CTRL_PWR_FLT;
      =     L 0.0;
      A     L 0.0;
      BLD   102;
      =     "MAIN_POWER_DB".MAIN_PWR_ON_CMD;
      A     L 0.0;
      FP    "MAIN_POWER_DB".PULSE_1;
      =     L 0.1;
      A     L 0.1;
      JNB   _001;
      L     0;
      T     "MAIN_POWER_DB".MAIN_PWR_FLT_TIMR;
_001: NOP   0;
      A     L 0.1;
      JNB   _002;
      L     0;
      T     "MAIN_POWER_DB".CTRL_PWR_FLT_TIMR;
_002: NOP   0;
NETWORK
TITLE =
      A     "ALWAYS_ON";
      =     L 0.0;
      A     L 0.0;
      A     "MAIN_POWER_DB".MAIN_PWR_ON_CMD;
      AN    "MAIN_POWER_DB".MAIN_PWR_ON_FB;
      AN    "MAIN_POWER_DB".MAIN_PWR_FLT;
      A     "ONE_SECOND_PULSE";
      JNB   _003;
      L     1;
      L     "MAIN_POWER_DB".MAIN_PWR_FLT_TIMR;
      +I;
      T     "MAIN_POWER_DB".MAIN_PWR_FLT_TIMR;
_003: NOP   0;
      A     L 0.0;
      A(;
      L     "MAIN_POWER_DB".MAIN_PWR_FLT_TIMR;
      L     3;
      >=I;
      );
      AN    "MAIN_POWER_DB".MAIN_PWR_ON_FB;
      =     "MAIN_POWER_DB".MAIN_PWR_FLT;
      A     L 0.0;
      A     "MAIN_POWER_DB".ALARM_ACK_PB;
      A     "MAIN_POWER_DB".MAIN_PWR_FLT;
      JNB   _004;
      L     0;
      T     "MAIN_POWER_DB".MAIN_PWR_FLT_TIMR;
_004: NOP   0;
NETWORK
TITLE =
      A     "ALWAYS_ON";
      A(;
      A     "MAIN_POWER_DB".MAIN_PWR_ON_CMD;
      A(;
      O     "MAIN_POWER_DB".MAIN_PWR_ON_FB;
      O     "HALF_SECOND_PULSE_TRAIN";
      );
      O     "MAIN_POWER_DB".LAMP_TEST_PB;
      );
      =     "MAIN_POWER_DB".MAIN_PWR_ON_IND;
NETWORK
TITLE =
      A     "ALWAYS_ON";
      A(;
      A     "MAIN_POWER_DB".MAIN_PWR_ON_CMD;
      A     "MAIN_POWER_DB".MAIN_PWR_ON_FB;
      A     "MAIN_POWER_DB".CTRL_PWR_ON_FB;
      O     "MAIN_POWER_DB".LAMP_TEST_PB;
      );
      =     "MAIN_POWER_DB".CTRL_PWR_ON_IND;
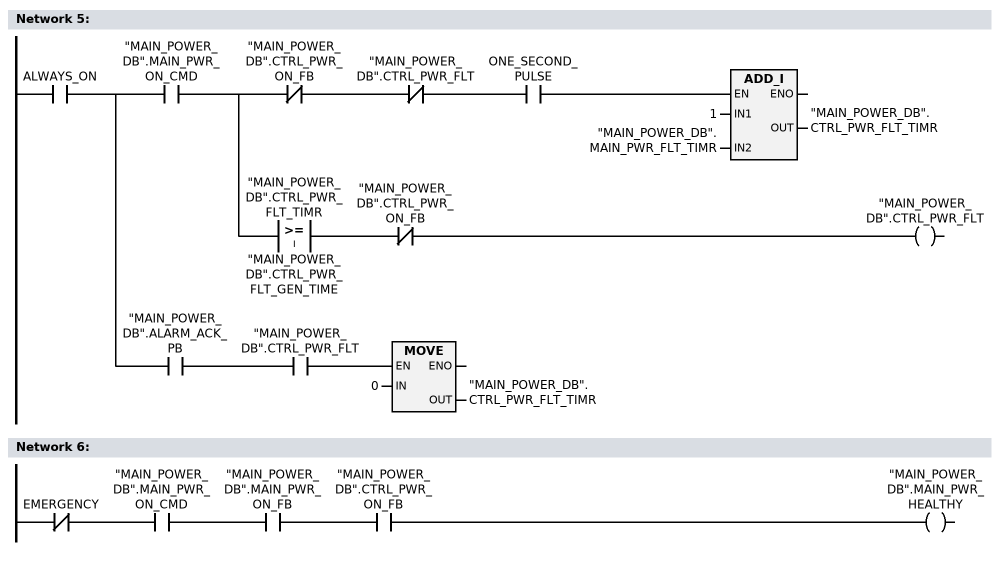
NETWORK
TITLE =
      A     "ALWAYS_ON";
      =     L 0.0;
      A     L 0.0;
      A     "MAIN_POWER_DB".MAIN_PWR_ON_CMD;
      =     L 0.1;
      A     L 0.1;
      AN    "MAIN_POWER_DB".CTRL_PWR_ON_FB;
      AN    "MAIN_POWER_DB".CTRL_PWR_FLT;
      A     "ONE_SECOND_PULSE";
      JNB   _005;
      L     1;
      L     "MAIN_POWER_DB".MAIN_PWR_FLT_TIMR;
      +I;
      T     "MAIN_POWER_DB".CTRL_PWR_FLT_TIMR;
_005: NOP   0;
      A     L 0.1;
      A(;
      L     "MAIN_POWER_DB".CTRL_PWR_FLT_TIMR;
      L     "MAIN_POWER_DB".CTRL_PWR_FLT_GEN_TIME;
      >=I;
      );
      AN    "MAIN_POWER_DB".CTRL_PWR_ON_FB;
      =     "MAIN_POWER_DB".CTRL_PWR_FLT;
      A     L 0.0;
      A     "MAIN_POWER_DB".ALARM_ACK_PB;
      A     "MAIN_POWER_DB".CTRL_PWR_FLT;
      JNB   _006;
      L     0;
      T     "MAIN_POWER_DB".CTRL_PWR_FLT_TIMR;
_006: NOP   0;
NETWORK
TITLE =
      AN    "EMERGENCY";
      A     "MAIN_POWER_DB".MAIN_PWR_ON_CMD;
      A     "MAIN_POWER_DB".MAIN_PWR_ON_FB;
      A     "MAIN_POWER_DB".CTRL_PWR_ON_FB;
      =     "MAIN_POWER_DB".MAIN_PWR_HEALTHY;
END_FUNCTION

FUNCTION "HYDRAULIC_SYSTEM" : VOID	// FC 4
AUTHOR : Kamillas
VERSION : 0.1
BEGIN
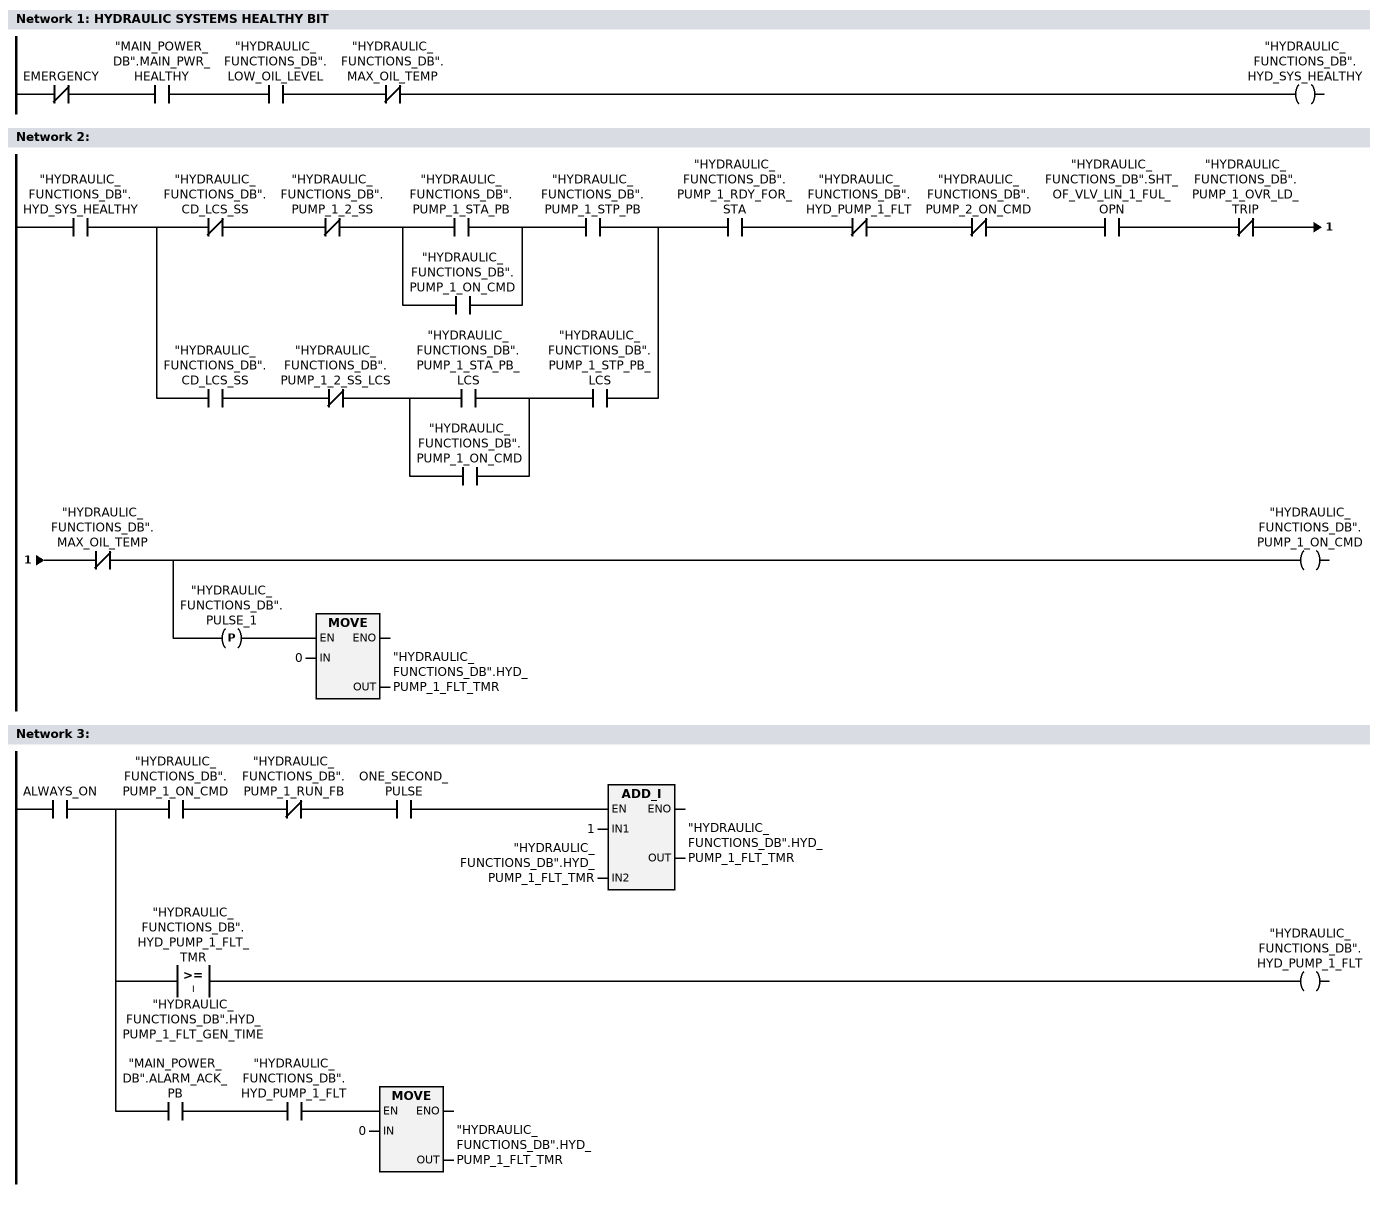
NETWORK
TITLE = HYDRAULIC SYSTEMS HEALTHY BIT
      AN    "EMERGENCY";
      A     "MAIN_POWER_DB".MAIN_PWR_HEALTHY;
      A     "HYDRAULIC_FUNCTIONS_DB".LOW_OIL_LEVEL;
      AN    "HYDRAULIC_FUNCTIONS_DB".MAX_OIL_TEMP;
      =     "HYDRAULIC_FUNCTIONS_DB".HYD_SYS_HEALTHY;
NETWORK
TITLE =
      A     "HYDRAULIC_FUNCTIONS_DB".HYD_SYS_HEALTHY;
      A(;
      AN    "HYDRAULIC_FUNCTIONS_DB".CD_LCS_SS;
      AN    "HYDRAULIC_FUNCTIONS_DB".PUMP_1_2_SS;
      A(;
      O     "HYDRAULIC_FUNCTIONS_DB".PUMP_1_STA_PB;
      O     "HYDRAULIC_FUNCTIONS_DB".PUMP_1_ON_CMD;
      );
      A     "HYDRAULIC_FUNCTIONS_DB".PUMP_1_STP_PB;
      O;
      A     "HYDRAULIC_FUNCTIONS_DB".CD_LCS_SS;
      AN    "HYDRAULIC_FUNCTIONS_DB".PUMP_1_2_SS_LCS;
      A(;
      O     "HYDRAULIC_FUNCTIONS_DB".PUMP_1_STA_PB_LCS;
      O     "HYDRAULIC_FUNCTIONS_DB".PUMP_1_ON_CMD;
      );
      A     "HYDRAULIC_FUNCTIONS_DB".PUMP_1_STP_PB_LCS;
      );
      A     "HYDRAULIC_FUNCTIONS_DB".PUMP_1_RDY_FOR_STA;
      AN    "HYDRAULIC_FUNCTIONS_DB".HYD_PUMP_1_FLT;
      AN    "HYDRAULIC_FUNCTIONS_DB".PUMP_2_ON_CMD;
      A     "HYDRAULIC_FUNCTIONS_DB".SHT_OF_VLV_LIN_1_FUL_OPN;
      AN    "HYDRAULIC_FUNCTIONS_DB".PUMP_1_OVR_LD_TRIP;
      AN    "HYDRAULIC_FUNCTIONS_DB".MAX_OIL_TEMP;
      =     L 0.0;
      A     L 0.0;
      BLD   102;
      =     "HYDRAULIC_FUNCTIONS_DB".PUMP_1_ON_CMD;
      A     L 0.0;
      FP    "HYDRAULIC_FUNCTIONS_DB".PULSE_1;
      JNB   _001;
      L     0;
      T     "HYDRAULIC_FUNCTIONS_DB".HYD_PUMP_1_FLT_TMR;
_001: NOP   0;
NETWORK
TITLE =
      A     "ALWAYS_ON";
      =     L 0.0;
      A     L 0.0;
      A     "HYDRAULIC_FUNCTIONS_DB".PUMP_1_ON_CMD;
      AN    "HYDRAULIC_FUNCTIONS_DB".PUMP_1_RUN_FB;
      A     "ONE_SECOND_PULSE";
      JNB   _002;
      L     1;
      L     "HYDRAULIC_FUNCTIONS_DB".HYD_PUMP_1_FLT_TMR;
      +I;
      T     "HYDRAULIC_FUNCTIONS_DB".HYD_PUMP_1_FLT_TMR;
_002: NOP   0;
      A     L 0.0;
      A(;
      L     "HYDRAULIC_FUNCTIONS_DB".HYD_PUMP_1_FLT_TMR;
      L     "HYDRAULIC_FUNCTIONS_DB".HYD_PUMP_1_FLT_GEN_TIME;
      >=I;
      );
      =     "HYDRAULIC_FUNCTIONS_DB".HYD_PUMP_1_FLT;
      A     L 0.0;
      A     "MAIN_POWER_DB".ALARM_ACK_PB;
      A     "HYDRAULIC_FUNCTIONS_DB".HYD_PUMP_1_FLT;
      JNB   _003;
      L     0;
      T     "HYDRAULIC_FUNCTIONS_DB".HYD_PUMP_1_FLT_TMR;
_003: NOP   0;
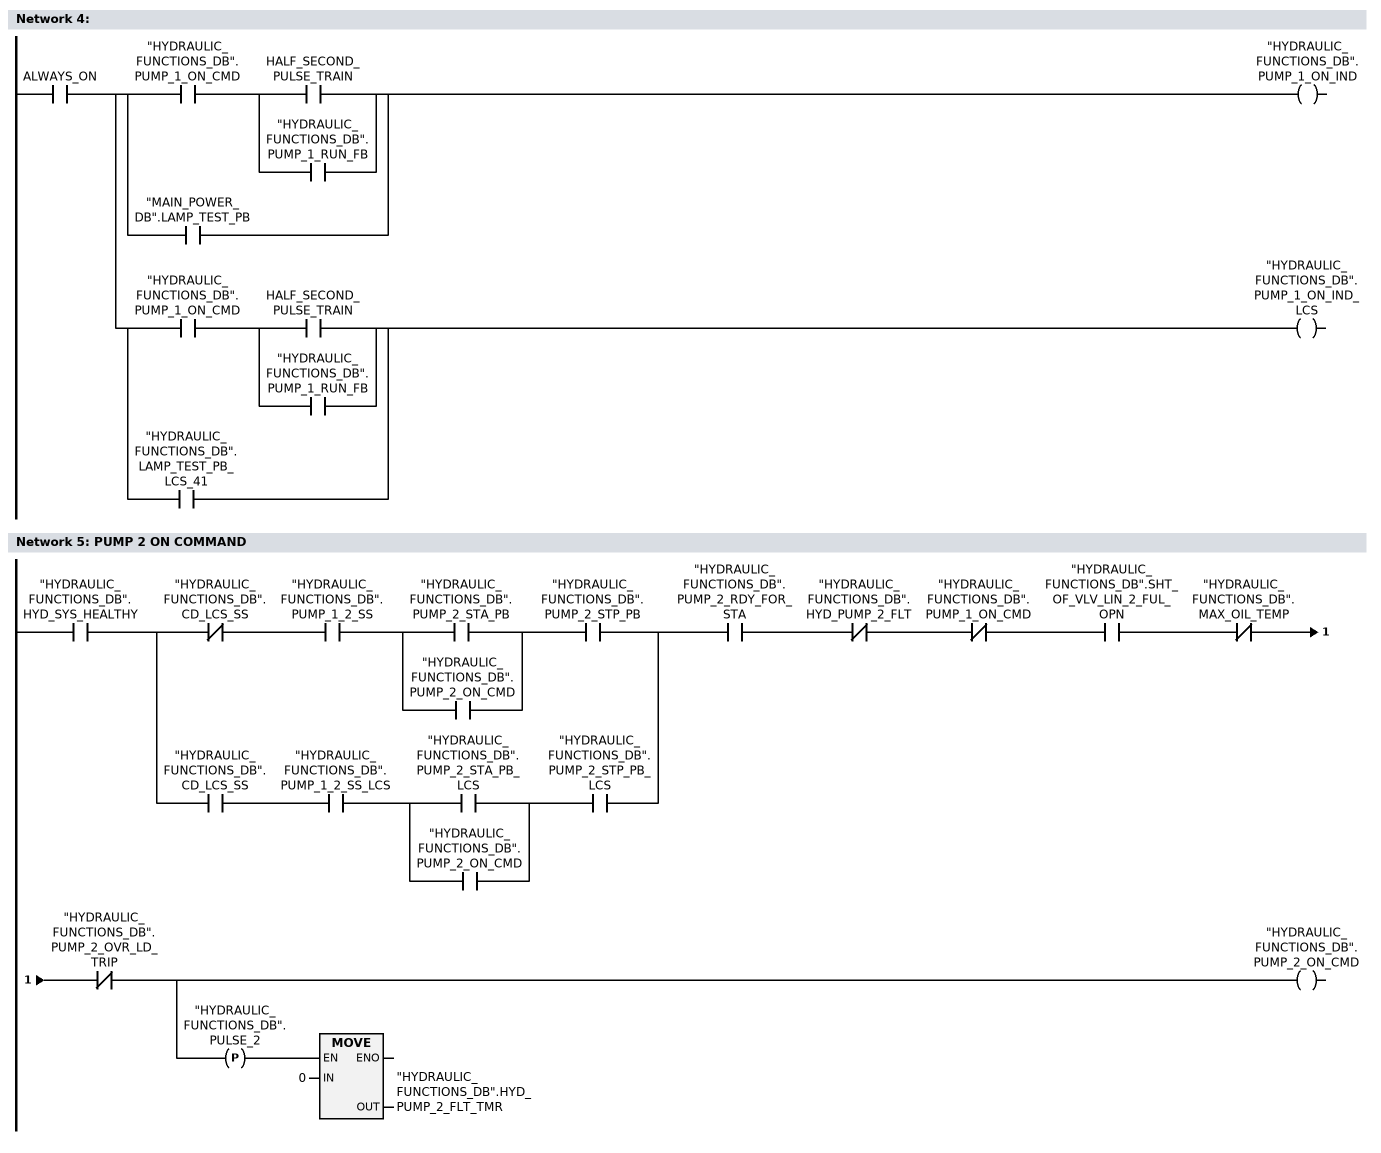
NETWORK
TITLE =
      A     "ALWAYS_ON";
      =     L 0.0;
      A     L 0.0;
      A(;
      A     "HYDRAULIC_FUNCTIONS_DB".PUMP_1_ON_CMD;
      A(;
      O     "HALF_SECOND_PULSE_TRAIN";
      O     "HYDRAULIC_FUNCTIONS_DB".PUMP_1_RUN_FB;
      );
      O     "MAIN_POWER_DB".LAMP_TEST_PB;
      );
      =     "HYDRAULIC_FUNCTIONS_DB".PUMP_1_ON_IND;
      A     L 0.0;
      A(;
      A     "HYDRAULIC_FUNCTIONS_DB".PUMP_1_ON_CMD;
      A(;
      O     "HALF_SECOND_PULSE_TRAIN";
      O     "HYDRAULIC_FUNCTIONS_DB".PUMP_1_RUN_FB;
      );
      O     "HYDRAULIC_FUNCTIONS_DB".LAMP_TEST_PB_LCS_41;
      );
      =     "HYDRAULIC_FUNCTIONS_DB".PUMP_1_ON_IND_LCS;
NETWORK
TITLE = PUMP 2 ON COMMAND
      A     "HYDRAULIC_FUNCTIONS_DB".HYD_SYS_HEALTHY;
      A(;
      AN    "HYDRAULIC_FUNCTIONS_DB".CD_LCS_SS;
      A     "HYDRAULIC_FUNCTIONS_DB".PUMP_1_2_SS;
      A(;
      O     "HYDRAULIC_FUNCTIONS_DB".PUMP_2_STA_PB;
      O     "HYDRAULIC_FUNCTIONS_DB".PUMP_2_ON_CMD;
      );
      A     "HYDRAULIC_FUNCTIONS_DB".PUMP_2_STP_PB;
      O;
      A     "HYDRAULIC_FUNCTIONS_DB".CD_LCS_SS;
      A     "HYDRAULIC_FUNCTIONS_DB".PUMP_1_2_SS_LCS;
      A(;
      O     "HYDRAULIC_FUNCTIONS_DB".PUMP_2_STA_PB_LCS;
      O     "HYDRAULIC_FUNCTIONS_DB".PUMP_2_ON_CMD;
      );
      A     "HYDRAULIC_FUNCTIONS_DB".PUMP_2_STP_PB_LCS;
      );
      A     "HYDRAULIC_FUNCTIONS_DB".PUMP_2_RDY_FOR_STA;
      AN    "HYDRAULIC_FUNCTIONS_DB".HYD_PUMP_2_FLT;
      AN    "HYDRAULIC_FUNCTIONS_DB".PUMP_1_ON_CMD;
      A     "HYDRAULIC_FUNCTIONS_DB".SHT_OF_VLV_LIN_2_FUL_OPN;
      AN    "HYDRAULIC_FUNCTIONS_DB".MAX_OIL_TEMP;
      AN    "HYDRAULIC_FUNCTIONS_DB".PUMP_2_OVR_LD_TRIP;
      =     L 0.0;
      A     L 0.0;
      BLD   102;
      =     "HYDRAULIC_FUNCTIONS_DB".PUMP_2_ON_CMD;
      A     L 0.0;
      FP    "HYDRAULIC_FUNCTIONS_DB".PULSE_2;
      JNB   _004;
      L     0;
      T     "HYDRAULIC_FUNCTIONS_DB".HYD_PUMP_2_FLT_TMR;
_004: NOP   0;
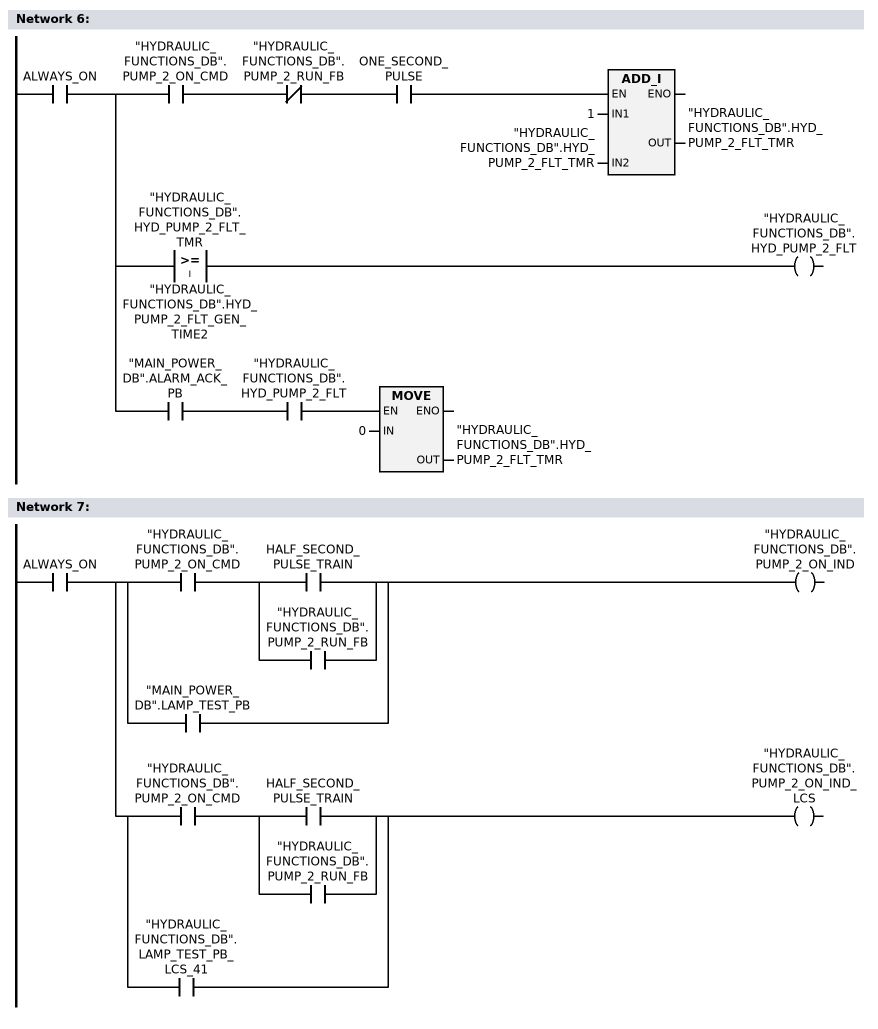
NETWORK
TITLE =
      A     "ALWAYS_ON";
      =     L 0.0;
      A     L 0.0;
      A     "HYDRAULIC_FUNCTIONS_DB".PUMP_2_ON_CMD;
      AN    "HYDRAULIC_FUNCTIONS_DB".PUMP_2_RUN_FB;
      A     "ONE_SECOND_PULSE";
      JNB   _005;
      L     1;
      L     "HYDRAULIC_FUNCTIONS_DB".HYD_PUMP_2_FLT_TMR;
      +I;
      T     "HYDRAULIC_FUNCTIONS_DB".HYD_PUMP_2_FLT_TMR;
_005: NOP   0;
      A     L 0.0;
      A(;
      L     "HYDRAULIC_FUNCTIONS_DB".HYD_PUMP_2_FLT_TMR;
      L     "HYDRAULIC_FUNCTIONS_DB".HYD_PUMP_2_FLT_GEN_TIME2;
      >=I;
      );
      =     "HYDRAULIC_FUNCTIONS_DB".HYD_PUMP_2_FLT;
      A     L 0.0;
      A     "MAIN_POWER_DB".ALARM_ACK_PB;
      A     "HYDRAULIC_FUNCTIONS_DB".HYD_PUMP_2_FLT;
      JNB   _006;
      L     0;
      T     "HYDRAULIC_FUNCTIONS_DB".HYD_PUMP_2_FLT_TMR;
_006: NOP   0;
NETWORK
TITLE =
      A     "ALWAYS_ON";
      =     L 0.0;
      A     L 0.0;
      A(;
      A     "HYDRAULIC_FUNCTIONS_DB".PUMP_2_ON_CMD;
      A(;
      O     "HALF_SECOND_PULSE_TRAIN";
      O     "HYDRAULIC_FUNCTIONS_DB".PUMP_2_RUN_FB;
      );
      O     "MAIN_POWER_DB".LAMP_TEST_PB;
      );
      =     "HYDRAULIC_FUNCTIONS_DB".PUMP_2_ON_IND;
      A     L 0.0;
      A(;
      A     "HYDRAULIC_FUNCTIONS_DB".PUMP_2_ON_CMD;
      A(;
      O     "HALF_SECOND_PULSE_TRAIN";
      O     "HYDRAULIC_FUNCTIONS_DB".PUMP_2_RUN_FB;
      );
      O     "HYDRAULIC_FUNCTIONS_DB".LAMP_TEST_PB_LCS_41;
      );
      =     "HYDRAULIC_FUNCTIONS_DB".PUMP_2_ON_IND_LCS;
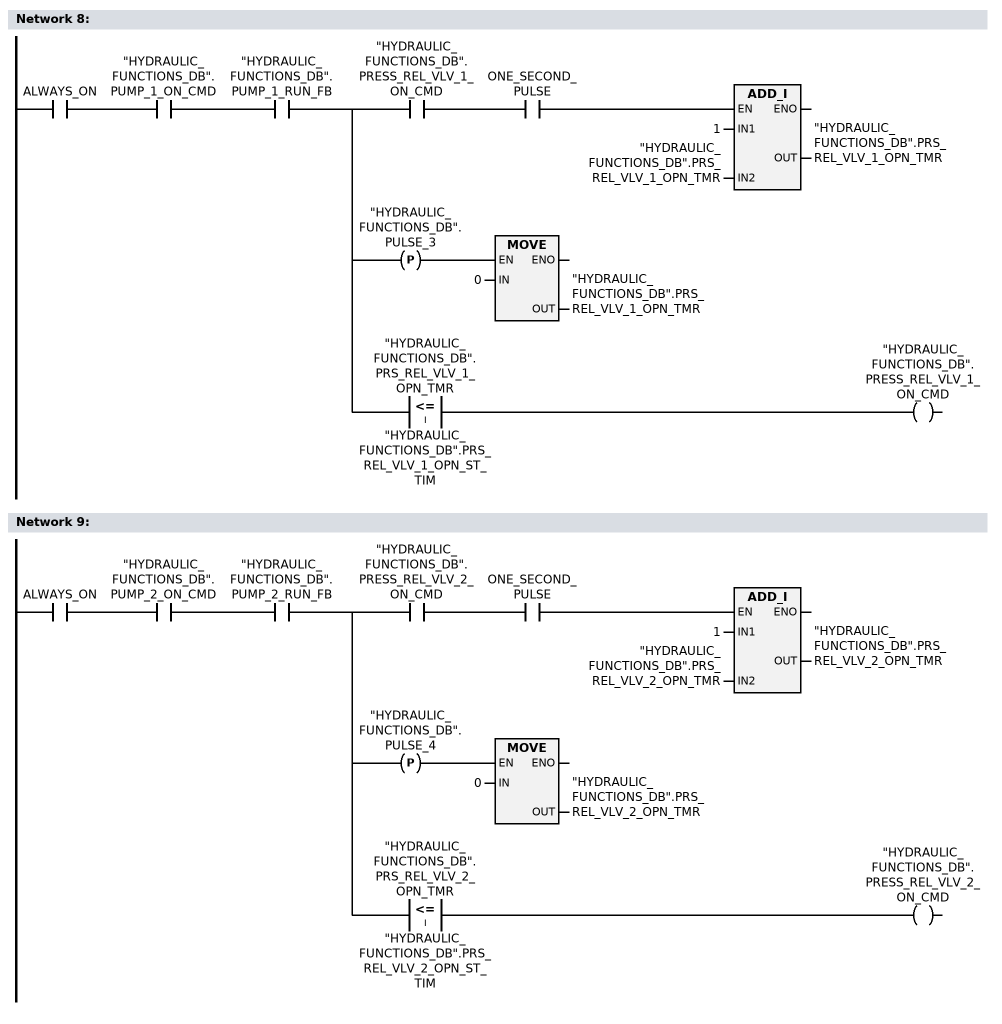
NETWORK
TITLE =
      A     "ALWAYS_ON";
      A     "HYDRAULIC_FUNCTIONS_DB".PUMP_1_ON_CMD;
      A     "HYDRAULIC_FUNCTIONS_DB".PUMP_1_RUN_FB;
      =     L 0.0;
      A     L 0.0;
      A     "HYDRAULIC_FUNCTIONS_DB".PRESS_REL_VLV_1_ON_CMD;
      A     "ONE_SECOND_PULSE";
      JNB   _007;
      L     1;
      L     "HYDRAULIC_FUNCTIONS_DB".PRS_REL_VLV_1_OPN_TMR;
      +I;
      T     "HYDRAULIC_FUNCTIONS_DB".PRS_REL_VLV_1_OPN_TMR;
_007: NOP   0;
      A     L 0.0;
      FP    "HYDRAULIC_FUNCTIONS_DB".PULSE_3;
      JNB   _008;
      L     0;
      T     "HYDRAULIC_FUNCTIONS_DB".PRS_REL_VLV_1_OPN_TMR;
_008: NOP   0;
      A     L 0.0;
      A(;
      L     "HYDRAULIC_FUNCTIONS_DB".PRS_REL_VLV_1_OPN_TMR;
      L     "HYDRAULIC_FUNCTIONS_DB".PRS_REL_VLV_1_OPN_ST_TIM;
      <=I;
      );
      =     "HYDRAULIC_FUNCTIONS_DB".PRESS_REL_VLV_1_ON_CMD;
NETWORK
TITLE =
      A     "ALWAYS_ON";
      A     "HYDRAULIC_FUNCTIONS_DB".PUMP_2_ON_CMD;
      A     "HYDRAULIC_FUNCTIONS_DB".PUMP_2_RUN_FB;
      =     L 0.0;
      A     L 0.0;
      A     "HYDRAULIC_FUNCTIONS_DB".PRESS_REL_VLV_2_ON_CMD;
      A     "ONE_SECOND_PULSE";
      JNB   _009;
      L     1;
      L     "HYDRAULIC_FUNCTIONS_DB".PRS_REL_VLV_2_OPN_TMR;
      +I;
      T     "HYDRAULIC_FUNCTIONS_DB".PRS_REL_VLV_2_OPN_TMR;
_009: NOP   0;
      A     L 0.0;
      FP    "HYDRAULIC_FUNCTIONS_DB".PULSE_4;
      JNB   _00a;
      L     0;
      T     "HYDRAULIC_FUNCTIONS_DB".PRS_REL_VLV_2_OPN_TMR;
_00a: NOP   0;
      A     L 0.0;
      A(;
      L     "HYDRAULIC_FUNCTIONS_DB".PRS_REL_VLV_2_OPN_TMR;
      L     "HYDRAULIC_FUNCTIONS_DB".PRS_REL_VLV_2_OPN_ST_TIM;
      <=I;
      );
      =     "HYDRAULIC_FUNCTIONS_DB".PRESS_REL_VLV_2_ON_CMD;
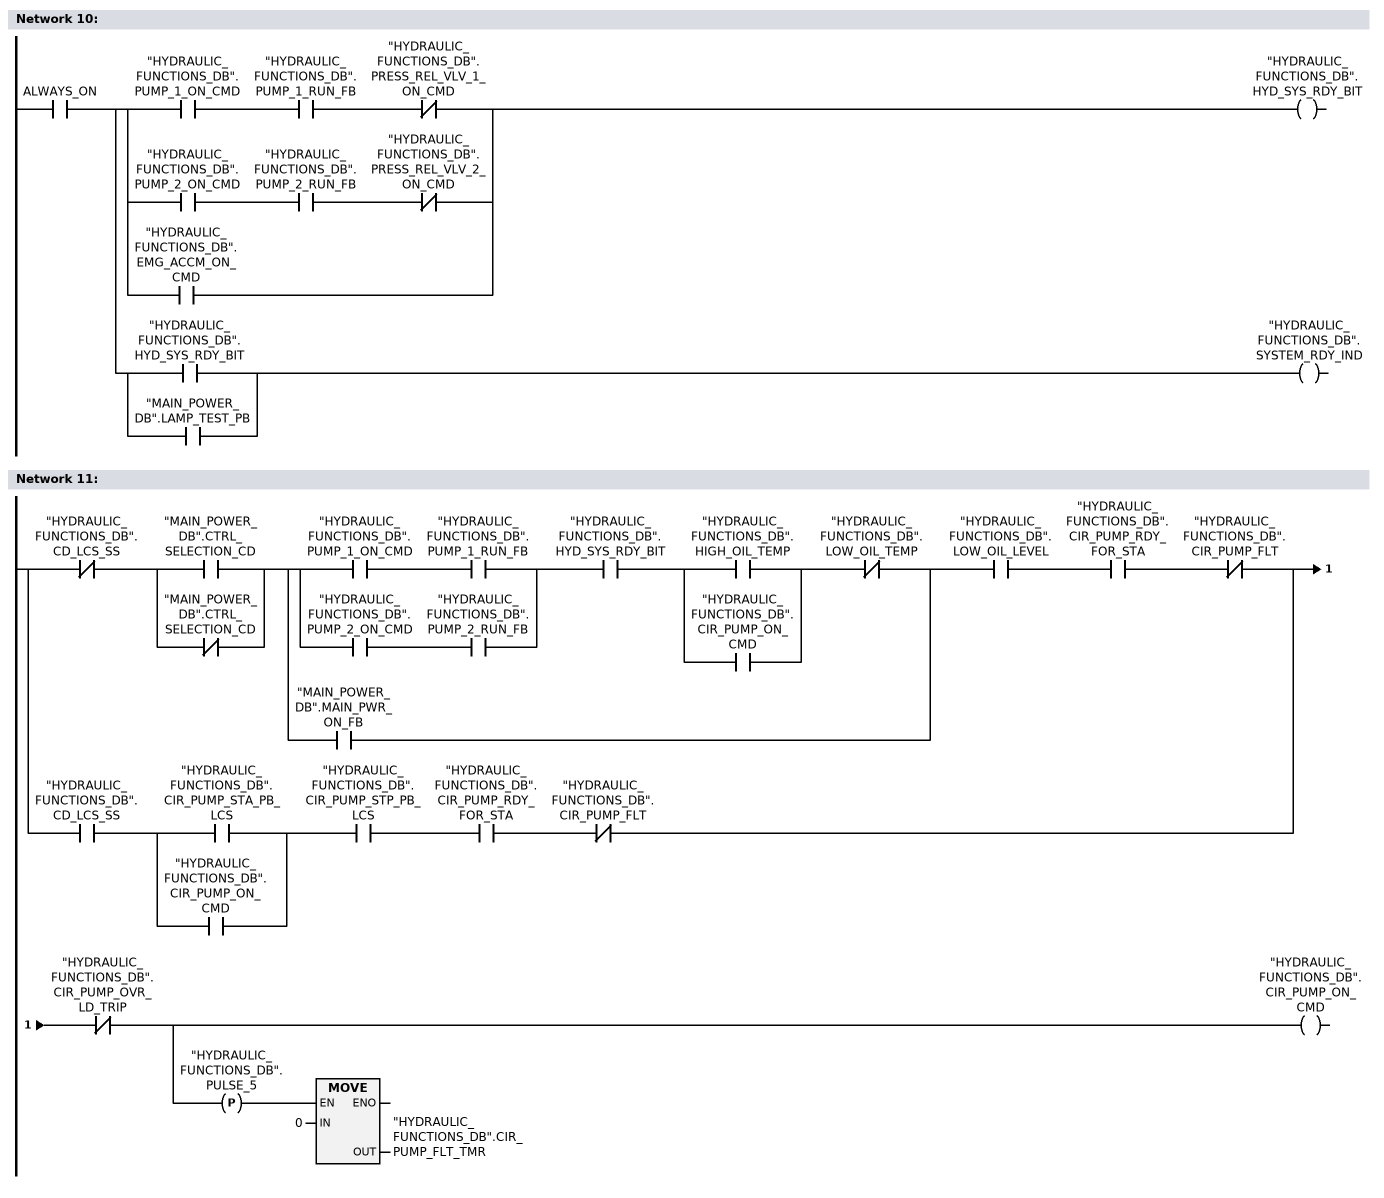
NETWORK
TITLE =
      A     "ALWAYS_ON";
      =     L 0.0;
      A     L 0.0;
      A(;
      A     "HYDRAULIC_FUNCTIONS_DB".PUMP_1_ON_CMD;
      A     "HYDRAULIC_FUNCTIONS_DB".PUMP_1_RUN_FB;
      AN    "HYDRAULIC_FUNCTIONS_DB".PRESS_REL_VLV_1_ON_CMD;
      O;
      A     "HYDRAULIC_FUNCTIONS_DB".PUMP_2_ON_CMD;
      A     "HYDRAULIC_FUNCTIONS_DB".PUMP_2_RUN_FB;
      AN    "HYDRAULIC_FUNCTIONS_DB".PRESS_REL_VLV_2_ON_CMD;
      O     "HYDRAULIC_FUNCTIONS_DB".EMG_ACCM_ON_CMD;
      );
      =     "HYDRAULIC_FUNCTIONS_DB".HYD_SYS_RDY_BIT;
      A     L 0.0;
      A(;
      O     "HYDRAULIC_FUNCTIONS_DB".HYD_SYS_RDY_BIT;
      O     "MAIN_POWER_DB".LAMP_TEST_PB;
      );
      =     "HYDRAULIC_FUNCTIONS_DB".SYSTEM_RDY_IND;
NETWORK
TITLE =
      A(;
      AN    "HYDRAULIC_FUNCTIONS_DB".CD_LCS_SS;
      A(;
      O     "MAIN_POWER_DB".CTRL_SELECTION_CD;
      ON    "MAIN_POWER_DB".CTRL_SELECTION_CD;
      );
      A(;
      A(;
      A     "HYDRAULIC_FUNCTIONS_DB".PUMP_1_ON_CMD;
      A     "HYDRAULIC_FUNCTIONS_DB".PUMP_1_RUN_FB;
      O;
      A     "HYDRAULIC_FUNCTIONS_DB".PUMP_2_ON_CMD;
      A     "HYDRAULIC_FUNCTIONS_DB".PUMP_2_RUN_FB;
      );
      A     "HYDRAULIC_FUNCTIONS_DB".HYD_SYS_RDY_BIT;
      A(;
      O     "HYDRAULIC_FUNCTIONS_DB".HIGH_OIL_TEMP;
      O     "HYDRAULIC_FUNCTIONS_DB".CIR_PUMP_ON_CMD;
      );
      AN    "HYDRAULIC_FUNCTIONS_DB".LOW_OIL_TEMP;
      O     "MAIN_POWER_DB".MAIN_PWR_ON_FB;
      );
      A     "HYDRAULIC_FUNCTIONS_DB".LOW_OIL_LEVEL;
      A     "HYDRAULIC_FUNCTIONS_DB".CIR_PUMP_RDY_FOR_STA;
      AN    "HYDRAULIC_FUNCTIONS_DB".CIR_PUMP_FLT;
      O;
      A     "HYDRAULIC_FUNCTIONS_DB".CD_LCS_SS;
      A(;
      O     "HYDRAULIC_FUNCTIONS_DB".CIR_PUMP_STA_PB_LCS;
      O     "HYDRAULIC_FUNCTIONS_DB".CIR_PUMP_ON_CMD;
      );
      A     "HYDRAULIC_FUNCTIONS_DB".CIR_PUMP_STP_PB_LCS;
      A     "HYDRAULIC_FUNCTIONS_DB".CIR_PUMP_RDY_FOR_STA;
      AN    "HYDRAULIC_FUNCTIONS_DB".CIR_PUMP_FLT;
      );
      AN    "HYDRAULIC_FUNCTIONS_DB".CIR_PUMP_OVR_LD_TRIP;
      =     L 0.0;
      A     L 0.0;
      BLD   102;
      =     "HYDRAULIC_FUNCTIONS_DB".CIR_PUMP_ON_CMD;
      A     L 0.0;
      FP    "HYDRAULIC_FUNCTIONS_DB".PULSE_5;
      JNB   _00b;
      L     0;
      T     "HYDRAULIC_FUNCTIONS_DB".CIR_PUMP_FLT_TMR;
_00b: NOP   0;
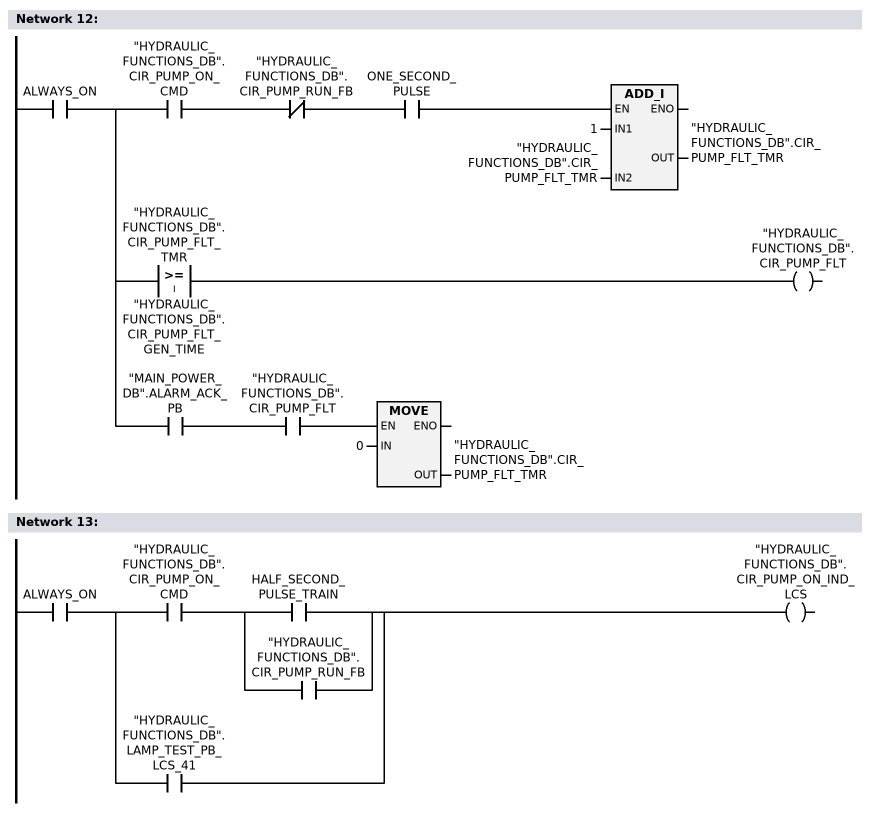
NETWORK
TITLE =
      A     "ALWAYS_ON";
      =     L 0.0;
      A     L 0.0;
      A     "HYDRAULIC_FUNCTIONS_DB".CIR_PUMP_ON_CMD;
      AN    "HYDRAULIC_FUNCTIONS_DB".CIR_PUMP_RUN_FB;
      A     "ONE_SECOND_PULSE";
      JNB   _00c;
      L     1;
      L     "HYDRAULIC_FUNCTIONS_DB".CIR_PUMP_FLT_TMR;
      +I;
      T     "HYDRAULIC_FUNCTIONS_DB".CIR_PUMP_FLT_TMR;
_00c: NOP   0;
      A     L 0.0;
      A(;
      L     "HYDRAULIC_FUNCTIONS_DB".CIR_PUMP_FLT_TMR;
      L     "HYDRAULIC_FUNCTIONS_DB".CIR_PUMP_FLT_GEN_TIME;
      >=I;
      );
      =     "HYDRAULIC_FUNCTIONS_DB".CIR_PUMP_FLT;
      A     L 0.0;
      A     "MAIN_POWER_DB".ALARM_ACK_PB;
      A     "HYDRAULIC_FUNCTIONS_DB".CIR_PUMP_FLT;
      JNB   _00d;
      L     0;
      T     "HYDRAULIC_FUNCTIONS_DB".CIR_PUMP_FLT_TMR;
_00d: NOP   0;
NETWORK
TITLE =
      A     "ALWAYS_ON";
      A(;
      A     "HYDRAULIC_FUNCTIONS_DB".CIR_PUMP_ON_CMD;
      A(;
      O     "HALF_SECOND_PULSE_TRAIN";
      O     "HYDRAULIC_FUNCTIONS_DB".CIR_PUMP_RUN_FB;
      );
      O     "HYDRAULIC_FUNCTIONS_DB".LAMP_TEST_PB_LCS_41;
      );
      =     "HYDRAULIC_FUNCTIONS_DB".CIR_PUMP_ON_IND_LCS;
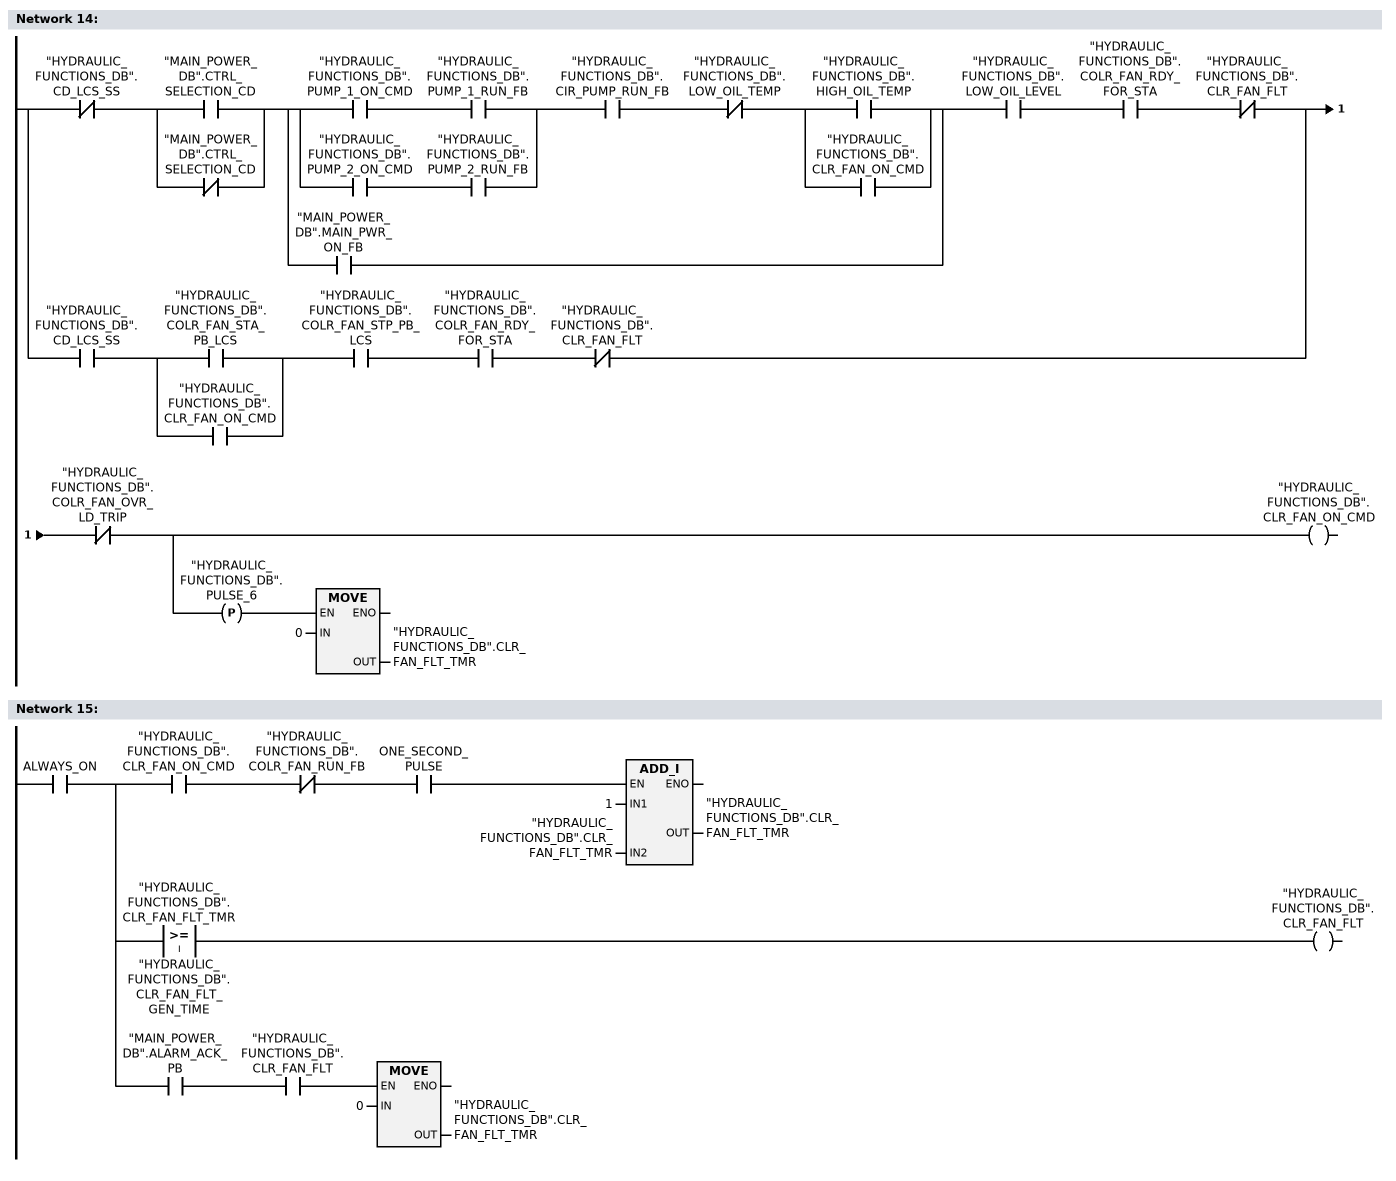
NETWORK
TITLE =
      A(;
      AN    "HYDRAULIC_FUNCTIONS_DB".CD_LCS_SS;
      A(;
      O     "MAIN_POWER_DB".CTRL_SELECTION_CD;
      ON    "MAIN_POWER_DB".CTRL_SELECTION_CD;
      );
      A(;
      A(;
      A     "HYDRAULIC_FUNCTIONS_DB".PUMP_1_ON_CMD;
      A     "HYDRAULIC_FUNCTIONS_DB".PUMP_1_RUN_FB;
      O;
      A     "HYDRAULIC_FUNCTIONS_DB".PUMP_2_ON_CMD;
      A     "HYDRAULIC_FUNCTIONS_DB".PUMP_2_RUN_FB;
      );
      A     "HYDRAULIC_FUNCTIONS_DB".CIR_PUMP_RUN_FB;
      AN    "HYDRAULIC_FUNCTIONS_DB".LOW_OIL_TEMP;
      A(;
      O     "HYDRAULIC_FUNCTIONS_DB".HIGH_OIL_TEMP;
      O     "HYDRAULIC_FUNCTIONS_DB".CLR_FAN_ON_CMD;
      );
      O     "MAIN_POWER_DB".MAIN_PWR_ON_FB;
      );
      A     "HYDRAULIC_FUNCTIONS_DB".LOW_OIL_LEVEL;
      A     "HYDRAULIC_FUNCTIONS_DB".COLR_FAN_RDY_FOR_STA;
      AN    "HYDRAULIC_FUNCTIONS_DB".CLR_FAN_FLT;
      O;
      A     "HYDRAULIC_FUNCTIONS_DB".CD_LCS_SS;
      A(;
      O     "HYDRAULIC_FUNCTIONS_DB".COLR_FAN_STA_PB_LCS;
      O     "HYDRAULIC_FUNCTIONS_DB".CLR_FAN_ON_CMD;
      );
      A     "HYDRAULIC_FUNCTIONS_DB".COLR_FAN_STP_PB_LCS;
      A     "HYDRAULIC_FUNCTIONS_DB".COLR_FAN_RDY_FOR_STA;
      AN    "HYDRAULIC_FUNCTIONS_DB".CLR_FAN_FLT;
      );
      AN    "HYDRAULIC_FUNCTIONS_DB".COLR_FAN_OVR_LD_TRIP;
      =     L 0.0;
      A     L 0.0;
      BLD   102;
      =     "HYDRAULIC_FUNCTIONS_DB".CLR_FAN_ON_CMD;
      A     L 0.0;
      FP    "HYDRAULIC_FUNCTIONS_DB".PULSE_6;
      JNB   _00e;
      L     0;
      T     "HYDRAULIC_FUNCTIONS_DB".CLR_FAN_FLT_TMR;
_00e: NOP   0;
NETWORK
TITLE =
      A     "ALWAYS_ON";
      =     L 0.0;
      A     L 0.0;
      A     "HYDRAULIC_FUNCTIONS_DB".CLR_FAN_ON_CMD;
      AN    "HYDRAULIC_FUNCTIONS_DB".COLR_FAN_RUN_FB;
      A     "ONE_SECOND_PULSE";
      JNB   _00f;
      L     1;
      L     "HYDRAULIC_FUNCTIONS_DB".CLR_FAN_FLT_TMR;
      +I;
      T     "HYDRAULIC_FUNCTIONS_DB".CLR_FAN_FLT_TMR;
_00f: NOP   0;
      A     L 0.0;
      A(;
      L     "HYDRAULIC_FUNCTIONS_DB".CLR_FAN_FLT_TMR;
      L     "HYDRAULIC_FUNCTIONS_DB".CLR_FAN_FLT_GEN_TIME;
      >=I;
      );
      =     "HYDRAULIC_FUNCTIONS_DB".CLR_FAN_FLT;
      A     L 0.0;
      A     "MAIN_POWER_DB".ALARM_ACK_PB;
      A     "HYDRAULIC_FUNCTIONS_DB".CLR_FAN_FLT;
      JNB   _010;
      L     0;
      T     "HYDRAULIC_FUNCTIONS_DB".CLR_FAN_FLT_TMR;
_010: NOP   0;
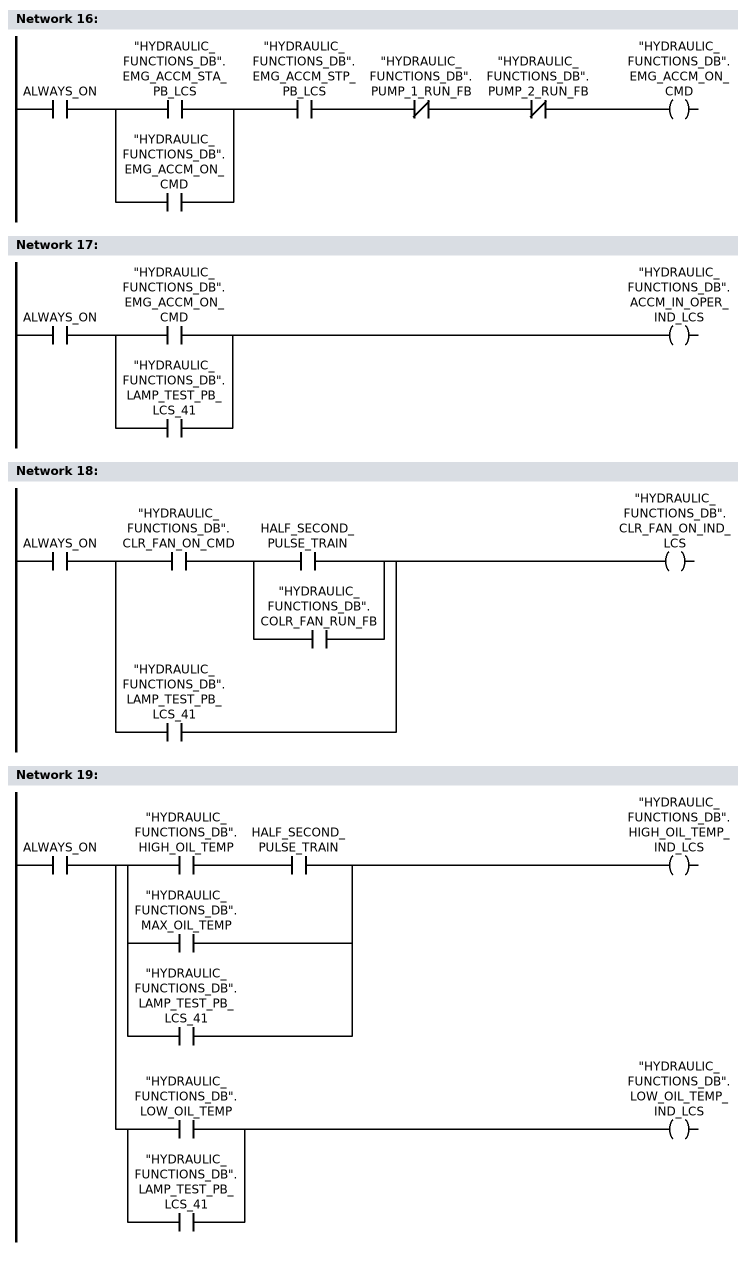
NETWORK
TITLE =
      A     "ALWAYS_ON";
      A(;
      O     "HYDRAULIC_FUNCTIONS_DB".EMG_ACCM_STA_PB_LCS;
      O     "HYDRAULIC_FUNCTIONS_DB".EMG_ACCM_ON_CMD;
      );
      A     "HYDRAULIC_FUNCTIONS_DB".EMG_ACCM_STP_PB_LCS;
      AN    "HYDRAULIC_FUNCTIONS_DB".PUMP_1_RUN_FB;
      AN    "HYDRAULIC_FUNCTIONS_DB".PUMP_2_RUN_FB;
      =     "HYDRAULIC_FUNCTIONS_DB".EMG_ACCM_ON_CMD;
NETWORK
TITLE =
      A     "ALWAYS_ON";
      A(;
      O     "HYDRAULIC_FUNCTIONS_DB".EMG_ACCM_ON_CMD;
      O     "HYDRAULIC_FUNCTIONS_DB".LAMP_TEST_PB_LCS_41;
      );
      =     "HYDRAULIC_FUNCTIONS_DB".ACCM_IN_OPER_IND_LCS;
NETWORK
TITLE =
      A     "ALWAYS_ON";
      A(;
      A     "HYDRAULIC_FUNCTIONS_DB".CLR_FAN_ON_CMD;
      A(;
      O     "HALF_SECOND_PULSE_TRAIN";
      O     "HYDRAULIC_FUNCTIONS_DB".COLR_FAN_RUN_FB;
      );
      O     "HYDRAULIC_FUNCTIONS_DB".LAMP_TEST_PB_LCS_41;
      );
      =     "HYDRAULIC_FUNCTIONS_DB".CLR_FAN_ON_IND_LCS;
NETWORK
TITLE =
      A     "ALWAYS_ON";
      =     L 0.0;
      A     L 0.0;
      A(;
      A     "HYDRAULIC_FUNCTIONS_DB".HIGH_OIL_TEMP;
      A     "HALF_SECOND_PULSE_TRAIN";
      O     "HYDRAULIC_FUNCTIONS_DB".MAX_OIL_TEMP;
      O     "HYDRAULIC_FUNCTIONS_DB".LAMP_TEST_PB_LCS_41;
      );
      =     "HYDRAULIC_FUNCTIONS_DB".HIGH_OIL_TEMP_IND_LCS;
      A     L 0.0;
      A(;
      O     "HYDRAULIC_FUNCTIONS_DB".LOW_OIL_TEMP;
      O     "HYDRAULIC_FUNCTIONS_DB".LAMP_TEST_PB_LCS_41;
      );
      =     "HYDRAULIC_FUNCTIONS_DB".LOW_OIL_TEMP_IND_LCS;
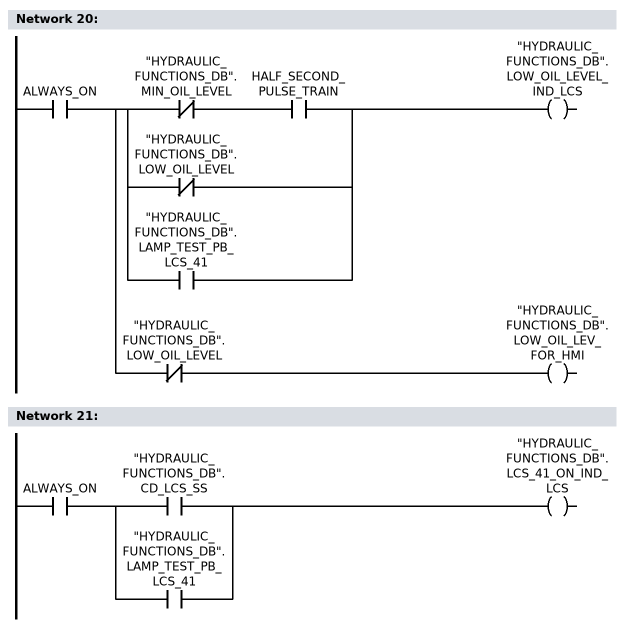
NETWORK
TITLE =
      A     "ALWAYS_ON";
      =     L 0.0;
      A     L 0.0;
      A(;
      AN    "HYDRAULIC_FUNCTIONS_DB".MIN_OIL_LEVEL;
      A     "HALF_SECOND_PULSE_TRAIN";
      ON    "HYDRAULIC_FUNCTIONS_DB".LOW_OIL_LEVEL;
      O     "HYDRAULIC_FUNCTIONS_DB".LAMP_TEST_PB_LCS_41;
      );
      =     "HYDRAULIC_FUNCTIONS_DB".LOW_OIL_LEVEL_IND_LCS;
      A     L 0.0;
      AN    "HYDRAULIC_FUNCTIONS_DB".LOW_OIL_LEVEL;
      =     "HYDRAULIC_FUNCTIONS_DB".LOW_OIL_LEV_FOR_HMI;
NETWORK
TITLE =
      A     "ALWAYS_ON";
      A(;
      O     "HYDRAULIC_FUNCTIONS_DB".CD_LCS_SS;
      O     "HYDRAULIC_FUNCTIONS_DB".LAMP_TEST_PB_LCS_41;
      );
      =     "HYDRAULIC_FUNCTIONS_DB".LCS_41_ON_IND_LCS;
END_FUNCTION

FUNCTION "LEVELLER_RAM" : VOID	// FC 5
AUTHOR : Kamillas
VERSION : 0.1
BEGIN
// (block stored without names or comments; labels and parameter names are numbered)
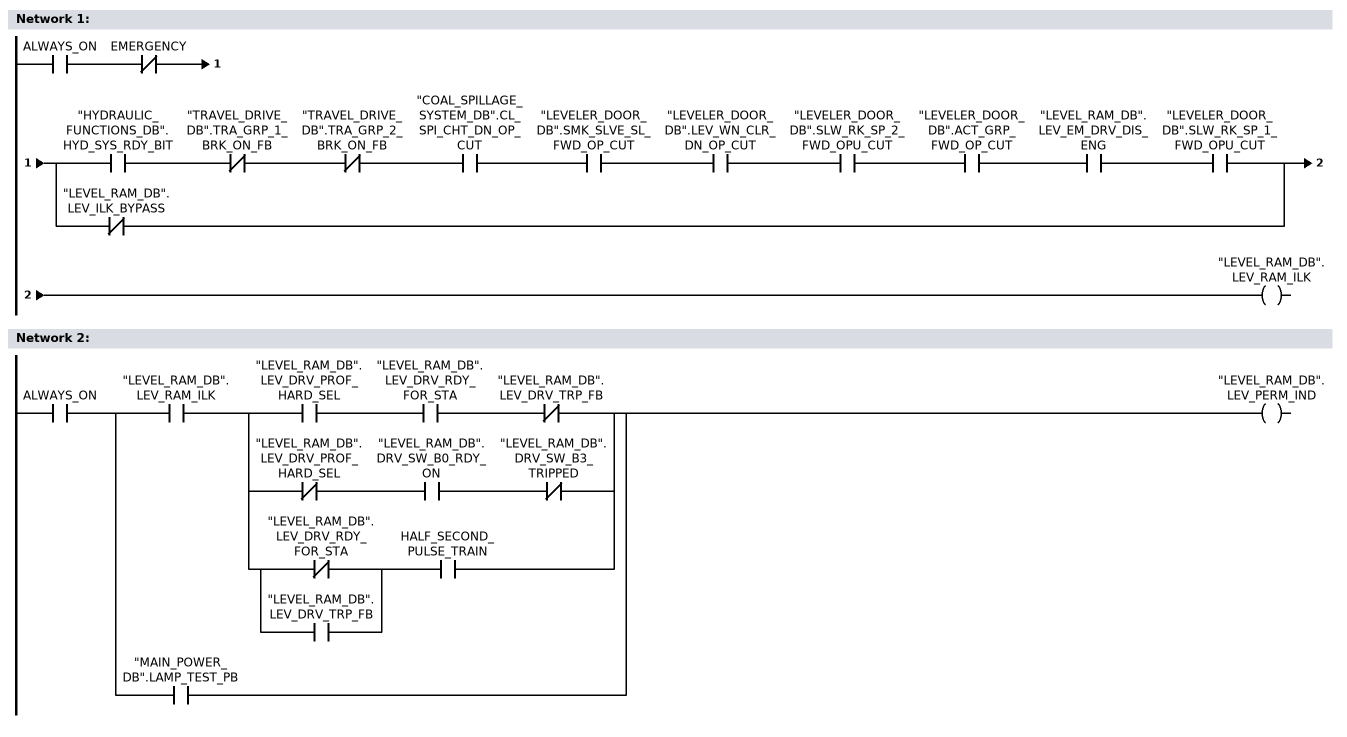
NETWORK
TITLE =
      A     "ALWAYS_ON";
      AN    "EMERGENCY";
      A(;
      A     "HYDRAULIC_FUNCTIONS_DB".HYD_SYS_RDY_BIT;
      AN    "TRAVEL_DRIVE_DB".TRA_GRP_1_BRK_ON_FB;
      AN    "TRAVEL_DRIVE_DB".TRA_GRP_2_BRK_ON_FB;
      A     "COAL_SPILLAGE_SYSTEM_DB".CL_SPI_CHT_DN_OP_CUT;
      A     "LEVELER_DOOR_DB".SMK_SLVE_SL_FWD_OP_CUT;
      A     "LEVELER_DOOR_DB".LEV_WN_CLR_DN_OP_CUT;
      A     "LEVELER_DOOR_DB".SLW_RK_SP_2_FWD_OPU_CUT;
      A     "LEVELER_DOOR_DB".ACT_GRP_FWD_OP_CUT;
      A     "LEVEL_RAM_DB".LEV_EM_DRV_DIS_ENG;
      A     "LEVELER_DOOR_DB".SLW_RK_SP_1_FWD_OPU_CUT;
      ON    "LEVEL_RAM_DB".LEV_ILK_BYPASS;
      );
      =     "LEVEL_RAM_DB".LEV_RAM_ILK;
NETWORK
TITLE =
      A     "ALWAYS_ON";
      A(;
      A     "LEVEL_RAM_DB".LEV_RAM_ILK;
      A(;
      A     "LEVEL_RAM_DB".LEV_DRV_PROF_HARD_SEL;
      A     "LEVEL_RAM_DB".LEV_DRV_RDY_FOR_STA;
      AN    "LEVEL_RAM_DB".LEV_DRV_TRP_FB;
      O;
      AN    "LEVEL_RAM_DB".LEV_DRV_PROF_HARD_SEL;
      A     "LEVEL_RAM_DB".DRV_SW_B0_RDY_ON;
      AN    "LEVEL_RAM_DB".DRV_SW_B3_TRIPPED;
      O;
      A(;
      ON    "LEVEL_RAM_DB".LEV_DRV_RDY_FOR_STA;
      O     "LEVEL_RAM_DB".LEV_DRV_TRP_FB;
      );
      A     "HALF_SECOND_PULSE_TRAIN";
      );
      O     "MAIN_POWER_DB".LAMP_TEST_PB;
      );
      =     "LEVEL_RAM_DB".LEV_PERM_IND;
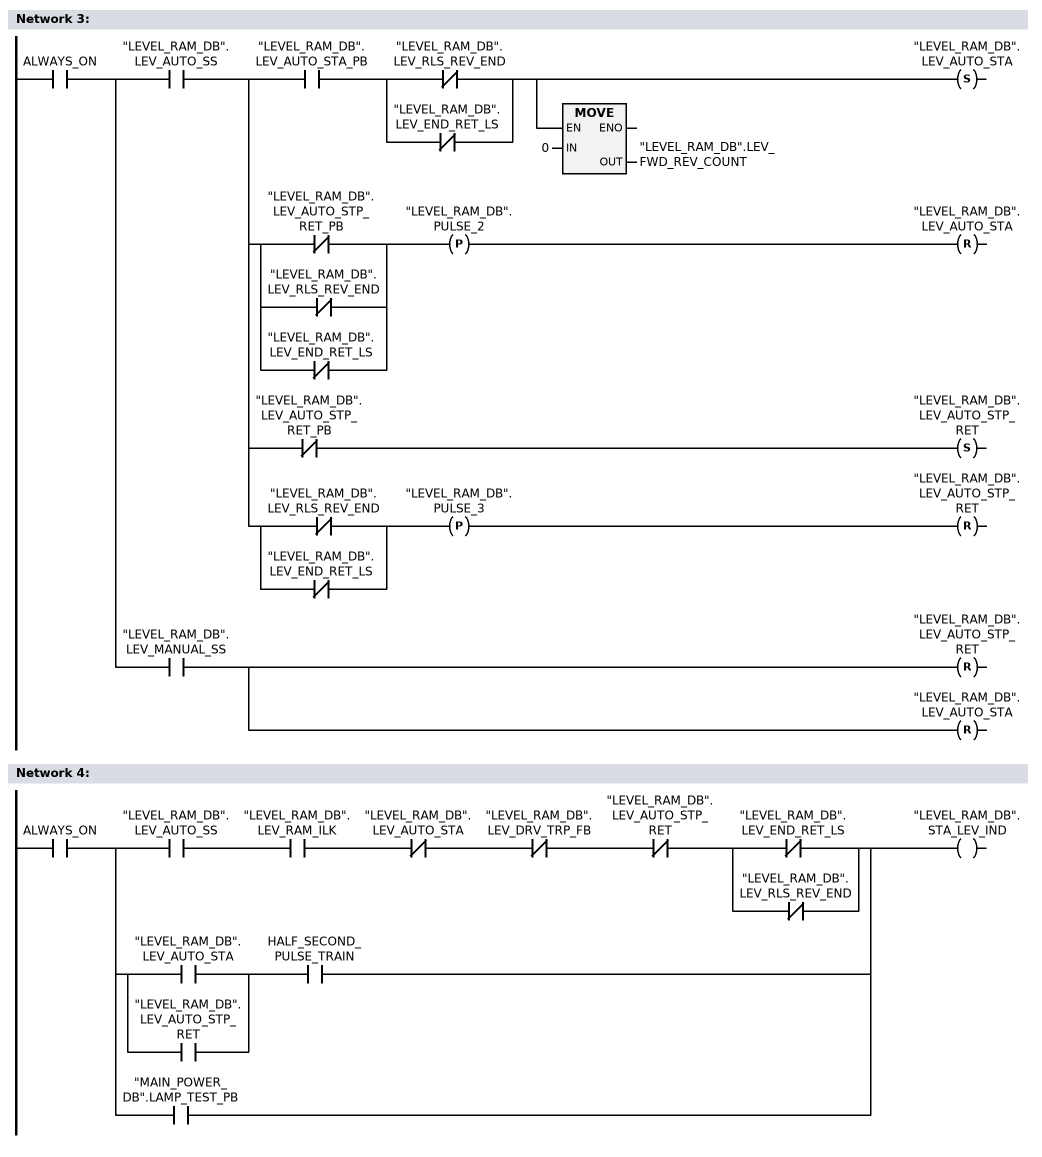
NETWORK
TITLE =
      A     "ALWAYS_ON";
      =     L 0.0;
      A     L 0.0;
      A     "LEVEL_RAM_DB".LEV_AUTO_SS;
      =     L 0.1;
      A     L 0.1;
      A     "LEVEL_RAM_DB".LEV_AUTO_STA_PB;
      A(;
      ON    "LEVEL_RAM_DB".LEV_RLS_REV_END;
      ON    "LEVEL_RAM_DB".LEV_END_RET_LS;
      );
      =     L 0.2;
      A     L 0.2;
      BLD   102;
      S     "LEVEL_RAM_DB".LEV_AUTO_STA;
      A     L 0.2;
      JNB   M001;
      L     0;
      T     "LEVEL_RAM_DB".LEV_FWD_REV_COUNT;
M001: NOP   0;
      A     L 0.1;
      A(;
      ON    "LEVEL_RAM_DB".LEV_AUTO_STP_RET_PB;
      ON    "LEVEL_RAM_DB".LEV_RLS_REV_END;
      ON    "LEVEL_RAM_DB".LEV_END_RET_LS;
      );
      FP    "LEVEL_RAM_DB".PULSE_2;
      R     "LEVEL_RAM_DB".LEV_AUTO_STA;
      A     L 0.1;
      AN    "LEVEL_RAM_DB".LEV_AUTO_STP_RET_PB;
      S     "LEVEL_RAM_DB".LEV_AUTO_STP_RET;
      A     L 0.1;
      A(;
      ON    "LEVEL_RAM_DB".LEV_RLS_REV_END;
      ON    "LEVEL_RAM_DB".LEV_END_RET_LS;
      );
      FP    "LEVEL_RAM_DB".PULSE_3;
      R     "LEVEL_RAM_DB".LEV_AUTO_STP_RET;
      A     L 0.0;
      A     "LEVEL_RAM_DB".LEV_MANUAL_SS;
      R     "LEVEL_RAM_DB".LEV_AUTO_STP_RET;
      R     "LEVEL_RAM_DB".LEV_AUTO_STA;
NETWORK
TITLE =
      A     "ALWAYS_ON";
      A(;
      A     "LEVEL_RAM_DB".LEV_AUTO_SS;
      A     "LEVEL_RAM_DB".LEV_RAM_ILK;
      AN    "LEVEL_RAM_DB".LEV_AUTO_STA;
      AN    "LEVEL_RAM_DB".LEV_DRV_TRP_FB;
      AN    "LEVEL_RAM_DB".LEV_AUTO_STP_RET;
      A(;
      ON    "LEVEL_RAM_DB".LEV_END_RET_LS;
      ON    "LEVEL_RAM_DB".LEV_RLS_REV_END;
      );
      O;
      A(;
      O     "LEVEL_RAM_DB".LEV_AUTO_STA;
      O     "LEVEL_RAM_DB".LEV_AUTO_STP_RET;
      );
      A     "HALF_SECOND_PULSE_TRAIN";
      O     "MAIN_POWER_DB".LAMP_TEST_PB;
      );
      =     "LEVEL_RAM_DB".STA_LEV_IND;
